LIN {X 0,Y 366.539,Z 659.329,A -85,B 0,C 180,E1 16261.22,E2 16261.22} C_VEL
LIN {X 0,Y 369.603,Z 643.731,A -85,B 0,C 180,E1 16259.522,E2 16259.522} C_VEL
LIN {X 0,Y 372.443,Z 626.719,A -85,B 0,C 180,E1 16258.031,E2 16258.031} C_VEL
LIN {X 0,Y 374.739,Z 609.542,A -85,B 0,C 180,E1 16256.842,E2 16256.842} C_VEL
LIN {X 0,Y 376.605,Z 590.744,A -85,B 0,C 180,E1 16255.852,E2 16255.852} C_VEL
LIN {X 0,Y 377.824,Z 571.243,A -85,B 0,C 180,E1 16255.127,E2 16255.127} C_VEL
LIN {X 0,Y 378.505,Z 547.045,A -85,B 0,C 180,E1 16254.58,E2 16254.58} C_VEL
LIN {X 0,Y 383.388,Z 388.518,A -85,B 0,C 180,E1 16251.66,E2 16251.66} C_VEL
LIN {X 0,Y 372.23,Z 368.985,A -85,B 0,C 180,E1 16249.629,E2 16249.629} C_VEL
LIN {X 0,Y 361.52,Z 352.259,A -85,B 0,C 180,E1 16247.541,E2 16247.541} C_VEL
LIN {X 0,Y 358.785,Z 347.938,A -85,B 0,C 180,E1 16246.899,E2 16246.899} C_VEL
LIN {X 0,Y 353.532,Z 335.825,A -85,B 0,C 180,E1 16243.861,E2 16243.861} C_VEL
LIN {X 0,Y 349.647,Z 327.602,A -85,B 0,C 180,E1 16241.563,E2 16241.563} C_VEL
LIN {X 0,Y 347.304,Z 322.978,A -85,B 0,C 180,E1 16240.157,E2 16240.157} C_VEL
LIN {X 0,Y 345.919,Z 319.541,A -85,B 0,C 180,E1 16239.059,E2 16239.059} C_VEL
LIN {X 0,Y 345.894,Z 319.384,A -85,B 0,C 180,E1 16234.823,E2 16234.823} C_VEL
LIN {X 0,Y 345.892,Z 319.382,A -85,B 0,C 180,E1 16230.527,E2 16230.527} C_VEL
LIN {X 0,Y 345.896,Z 319.388,A -85,B 0,C 180,E1 16226.354,E2 16226.354} C_VEL
LIN {X 0,Y 345.893,Z 319.4,A -85,B 0,C 180,E1 16222.252,E2 16222.252} C_VEL
LIN {X 0,Y 345.899,Z 319.385,A -85,B 0,C 180,E1 16218.014,E2 16218.014} C_VEL
LIN {X 0,Y 345.906,Z 319.366,A -85,B 0,C 180,E1 16213.785,E2 16213.785} C_VEL
LIN {X 0,Y 345.898,Z 319.37,A -85,B 0,C 180,E1 16209.484,E2 16209.484} C_VEL
LIN {X 0,Y 345.89,Z 319.398,A -85,B 0,C 180,E1 16205.308,E2 16205.308} C_VEL
LIN {X 0,Y 345.877,Z 319.386,A -85,B 0,C 180,E1 16201.16,E2 16201.16} C_VEL
LIN {X 0,Y 345.871,Z 319.369,A -85,B 0,C 180,E1 16197.018,E2 16197.018} C_VEL
LIN {X 0,Y 345.87,Z 319.378,A -85,B 0,C 180,E1 16192.86,E2 16192.86} C_VEL
LIN {X 0,Y 345.873,Z 319.401,A -85,B 0,C 180,E1 16188.664,E2 16188.664} C_VEL
LIN {X 0,Y 345.873,Z 319.4,A -85,B 0,C 180,E1 16184.405,E2 16184.405} C_VEL
LIN {X 0,Y 345.88,Z 319.39,A -85,B 0,C 180,E1 16180.056,E2 16180.056} C_VEL
LIN {X 0,Y 345.886,Z 319.384,A -85,B 0,C 180,E1 16175.947,E2 16175.947} C_VEL
LIN {X 0,Y 345.901,Z 319.385,A -85,B 0,C 180,E1 16171.702,E2 16171.702} C_VEL
LIN {X 0,Y 345.947,Z 319.628,A -85,B 0,C 180,E1 16169.507,E2 16169.507} C_VEL
LIN {X 0,Y 347.584,Z 323.392,A -85,B 0,C 180,E1 16168.43,E2 16168.43} C_VEL
LIN {X 0,Y 348.628,Z 324.913,A -85,B 0,C 180,E1 16167.956,E2 16167.956} C_VEL
LIN {X 0,Y 353.831,Z 334.918,A -85,B 0,C 180,E1 16165.39,E2 16165.39} C_VEL
LIN {X 0,Y 357.949,Z 342.981,A -85,B 0,C 180,E1 16163.49,E2 16163.49} C_VEL
LIN {X 0,Y 364.694,Z 357.152,A -85,B 0,C 180,E1 16160.502,E2 16160.502} C_VEL
LIN {X 0,Y 371.956,Z 374.258,A -85,B 0,C 180,E1 16157.359,E2 16157.359} C_VEL
LIN {X 0,Y 374.056,Z 379.335,A -85,B 0,C 180,E1 16156.557,E2 16156.557} C_VEL
LIN {X 0,Y 381.034,Z 392.431,A -85,B 0,C 180,E1 16155.246,E2 16155.246} C_VEL
LIN {X 0,Y 383.985,Z 429.126,A -85,B 0,C 180,E1 16153.918,E2 16153.918} C_VEL
LIN {X 0,Y 375.667,Z 632.493,A -85,B 0,C 180,E1 16149.71,E2 16149.71} C_VEL
LIN {X 0,Y 373.709,Z 654.478,A -85,B 0,C 180,E1 16149.004,E2 16149.004} C_VEL
LIN {X 0,Y 371.041,Z 675.386,A -85,B 0,C 180,E1 16148.054,E2 16148.054} C_VEL
LIN {X 0,Y 368.083,Z 694.62,A -85,B 0,C 180,E1 16146.892,E2 16146.892} C_VEL
LIN {X 0,Y 364.802,Z 713.742,A -85,B 0,C 180,E1 16145.427,E2 16145.427} C_VEL
LIN {X 0,Y 361.389,Z 732.08,A -85,B 0,C 180,E1 16143.691,E2 16143.691} C_VEL
LIN {X 0,Y 357.817,Z 750.227,A -85,B 0,C 180,E1 16141.596,E2 16141.596} C_VEL
LIN {X 0,Y 354.467,Z 767.276,A -85,B 0,C 180,E1 16139.207,E2 16139.207} C_VEL
LIN {X 0,Y 351.414,Z 783.149,A -85,B 0,C 180,E1 16136.531,E2 16136.531} C_VEL
LIN {X 0,Y 348.903,Z 797.366,A -85,B 0,C 180,E1 16133.653,E2 16133.653} C_VEL
LIN {X 0,Y 346.99,Z 809.978,A -85,B 0,C 180,E1 16130.581,E2 16130.581} C_VEL
LIN {X 0,Y 345.729,Z 820.44,A -85,B 0,C 180,E1 16127.503,E2 16127.503} C_VEL
LIN {X 0,Y 345.044,Z 829.017,A -85,B 0,C 180,E1 16124.43,E2 16124.43} C_VEL
LIN {X 0,Y 344.787,Z 836.104,A -85,B 0,C 180,E1 16121.203,E2 16121.203} C_VEL
LIN {X 0,Y 344.85,Z 841.123,A -85,B 0,C 180,E1 16118.167,E2 16118.167} C_VEL
LIN {X 0,Y 345.058,Z 844.743,A -85,B 0,C 180,E1 16114.987,E2 16114.987} C_VEL
LIN {X 0,Y 345.211,Z 846.508,A -85,B 0,C 180,E1 16112.158,E2 16112.158} C_VEL
LIN {X 0,Y 345.255,Z 846.827,A -85,B 0,C 180,E1 16109.17,E2 16109.17} C_VEL
LIN {X 0,Y 345.126,Z 845.656,A -85,B 0,C 180,E1 16106.179,E2 16106.179} C_VEL
LIN {X 0,Y 344.931,Z 842.863,A -85,B 0,C 180,E1 16103.175,E2 16103.175} C_VEL
LIN {X 0,Y 344.793,Z 838.223,A -85,B 0,C 180,E1 16099.98,E2 16099.98} C_VEL
LIN {X 0,Y 344.896,Z 831.799,A -85,B 0,C 180,E1 16096.761,E2 16096.761} C_VEL
LIN {X 0,Y 345.408,Z 823.997,A -85,B 0,C 180,E1 16093.693,E2 16093.693} C_VEL
LIN {X 0,Y 346.494,Z 813.722,A -85,B 0,C 180,E1 16090.444,E2 16090.444} C_VEL
LIN {X 0,Y 348.173,Z 801.841,A -85,B 0,C 180,E1 16087.369,E2 16087.369} C_VEL
LIN {X 0,Y 350.447,Z 788.441,A -85,B 0,C 180,E1 16084.481,E2 16084.481} C_VEL
LIN {X 0,Y 353.14,Z 774.009,A -85,B 0,C 180,E1 16081.874,E2 16081.874} C_VEL
LIN {X 0,Y 356.244,Z 758.161,A -85,B 0,C 180,E1 16079.47,E2 16079.47} C_VEL
LIN {X 0,Y 359.673,Z 740.767,A -85,B 0,C 180,E1 16077.27,E2 16077.27} C_VEL
LIN {X 0,Y 363.194,Z 722.371,A -85,B 0,C 180,E1 16075.356,E2 16075.356} C_VEL
LIN {X 0,Y 366.647,Z 702.966,A -85,B 0,C 180,E1 16073.719,E2 16073.719} C_VEL
LIN {X 0,Y 369.743,Z 683.735,A -85,B 0,C 180,E1 16072.426,E2 16072.426} C_VEL
LIN {X 0,Y 372.564,Z 663.659,A -85,B 0,C 180,E1 16071.389,E2 16071.389} C_VEL
LIN {X 0,Y 374.836,Z 642.783,A -85,B 0,C 180,E1 16070.598,E2 16070.598} C_VEL
LIN {X 0,Y 376.217,Z 620.758,A -85,B 0,C 180,E1 16070.027,E2 16070.027} C_VEL
LIN {X 0,Y 383.944,Z 427.198,A -85,B 0,C 180,E1 16066.047,E2 16066.047} C_VEL
LIN {X 0,Y 380.702,Z 391.532,A -85,B 0,C 180,E1 16064.711,E2 16064.711} C_VEL
LIN {X 0,Y 373.38,Z 377.914,A -85,B 0,C 180,E1 16063.277,E2 16063.277} C_VEL
LIN {X 0,Y 366.854,Z 362.006,A -85,B 0,C 180,E1 16060.441,E2 16060.441} C_VEL
LIN {X 0,Y 360.67,Z 348.666,A -85,B 0,C 180,E1 16057.782,E2 16057.782} C_VEL
LIN {X 0,Y 355.146,Z 337.373,A -85,B 0,C 180,E1 16055.25,E2 16055.25} C_VEL
LIN {X 0,Y 350.284,Z 328.233,A -85,B 0,C 180,E1 16052.947,E2 16052.947} C_VEL
LIN {X 0,Y 348.264,Z 324.159,A -85,B 0,C 180,E1 16051.888,E2 16051.888} C_VEL
LIN {X 0,Y 346.287,Z 320.952,A -85,B 0,C 180,E1 16050.927,E2 16050.927} C_VEL
LIN {X 0,Y 345.918,Z 319.456,A -85,B 0,C 180,E1 16050.413,E2 16050.413} C_VEL
LIN {X 0,Y 345.898,Z 319.385,A -85,B 0,C 180,E1 16046.248,E2 16046.248} C_VEL
LIN {X 0,Y 345.886,Z 319.383,A -85,B 0,C 180,E1 16042.073,E2 16042.073} C_VEL
LIN {X 0,Y 345.877,Z 319.378,A -85,B 0,C 180,E1 16037.844,E2 16037.844} C_VEL
LIN {X 0,Y 345.87,Z 319.372,A -85,B 0,C 180,E1 16033.542,E2 16033.542} C_VEL
LIN {X 0,Y 345.87,Z 319.379,A -85,B 0,C 180,E1 16029.316,E2 16029.316} C_VEL
LIN {X 0,Y 345.873,Z 319.402,A -85,B 0,C 180,E1 16025.141,E2 16025.141} C_VEL
LIN {X 0,Y 345.872,Z 319.39,A -85,B 0,C 180,E1 16020.993,E2 16020.993} C_VEL
LIN {X 0,Y 345.87,Z 319.369,A -85,B 0,C 180,E1 16016.851,E2 16016.851} C_VEL
LIN {X 0,Y 345.884,Z 319.379,A -85,B 0,C 180,E1 16012.692,E2 16012.692} C_VEL
LIN {X 0,Y 345.897,Z 319.401,A -85,B 0,C 180,E1 16008.491,E2 16008.491} C_VEL
LIN {X 0,Y 345.908,Z 319.379,A -85,B 0,C 180,E1 16004.234,E2 16004.234} C_VEL
LIN {X 0,Y 345.896,Z 319.37,A -85,B 0,C 180,E1 15999.956,E2 15999.956} C_VEL
LIN {X 0,Y 345.902,Z 319.373,A -85,B 0,C 180,E1 15995.947,E2 15995.947} C_VEL
LIN {X 0,Y 345.896,Z 319.385,A -85,B 0,C 180,E1 15991.701,E2 15991.701} C_VEL
LIN {X 0,Y 345.897,Z 319.393,A -85,B 0,C 180,E1 15987.569,E2 15987.569} C_VEL
LIN {X 0,Y 345.896,Z 319.393,A -85,B 0,C 180,E1 15983.453,E2 15983.453} C_VEL
LIN {X 0,Y 345.937,Z 319.68,A -85,B 0,C 180,E1 15980.73,E2 15980.73} C_VEL
LIN {X 0,Y 347.422,Z 323.162,A -85,B 0,C 180,E1 15979.643,E2 15979.643} C_VEL
LIN {X 0,Y 348.545,Z 325.55,A -85,B 0,C 180,E1 15978.934,E2 15978.934} C_VEL
LIN {X 0,Y 350.596,Z 329.771,A -85,B 0,C 180,E1 15977.697,E2 15977.697} C_VEL
LIN {X 0,Y 354.243,Z 337.521,A -85,B 0,C 180,E1 15975.568,E2 15975.568} C_VEL
LIN {X 0,Y 358.954,Z 348.373,A -85,B 0,C 180,E1 15972.896,E2 15972.896} C_VEL
LIN {X 0,Y 369.652,Z 364.898,A -85,B 0,C 180,E1 15970.738,E2 15970.738} C_VEL
LIN {X 0,Y 379.94,Z 382.361,A -85,B 0,C 180,E1 15968.834,E2 15968.834} C_VEL
LIN {X 0,Y 383.444,Z 389.074,A -85,B 0,C 180,E1 15968.206,E2 15968.206} C_VEL
LIN {X 0,Y 378.018,Z 564.942,A -85,B 0,C 180,E1 15964.946,E2 15964.946} C_VEL
LIN {X 0,Y 377.086,Z 583.644,A -85,B 0,C 180,E1 15964.345,E2 15964.345} C_VEL
LIN {X 0,Y 375.513,Z 601.927,A -85,B 0,C 180,E1 15963.496,E2 15963.496} C_VEL
LIN {X 0,Y 373.525,Z 618.693,A -85,B 0,C 180,E1 15962.458,E2 15962.458} C_VEL
LIN {X 0,Y 370.899,Z 636.019,A -85,B 0,C 180,E1 15961.094,E2 15961.094} C_VEL
LIN {X 0,Y 367.89,Z 652.482,A -85,B 0,C 180,E1 15959.466,E2 15959.466} C_VEL
LIN {X 0,Y 364.669,Z 667.723,A -85,B 0,C 180,E1 15957.604,E2 15957.604} C_VEL
LIN {X 0,Y 361.466,Z 681.388,A -85,B 0,C 180,E1 15955.563,E2 15955.563} C_VEL
LIN {X 0,Y 358.145,Z 694.464,A -85,B 0,C 180,E1 15953.18,E2 15953.18} C_VEL
LIN {X 0,Y 355.074,Z 705.939,A -85,B 0,C 180,E1 15950.608,E2 15950.608} C_VEL
LIN {X 0,Y 352.38,Z 715.885,A -85,B 0,C 180,E1 15947.845,E2 15947.845} C_VEL
LIN {X 0,Y 350.093,Z 724.318,A -85,B 0,C 180,E1 15944.894,E2 15944.894} C_VEL
LIN {X 0,Y 348.354,Z 731.066,A -85,B 0,C 180,E1 15941.831,E2 15941.831} C_VEL
LIN {X 0,Y 347.117,Z 736.256,A -85,B 0,C 180,E1 15938.614,E2 15938.614} C_VEL
LIN {X 0,Y 346.367,Z 739.644,A -85,B 0,C 180,E1 15935.466,E2 15935.466} C_VEL
LIN {X 0,Y 345.992,Z 741.548,A -85,B 0,C 180,E1 15932.153,E2 15932.153} C_VEL
LIN {X 0,Y 345.939,Z 741.818,A -85,B 0,C 180,E1 15928.841,E2 15928.841} C_VEL
LIN {X 0,Y 346.204,Z 740.465,A -85,B 0,C 180,E1 15925.528,E2 15925.528} C_VEL
LIN {X 0,Y 346.714,Z 738.05,A -85,B 0,C 180,E1 15922.764,E2 15922.764} C_VEL
LIN {X 0,Y 346.061,Z 736.752,A -85,B 0,C 180,E1 15921.504,E2 15921.504} C_VEL
LIN {X 0,Y 341.253,Z 732.89,A -85,B 0,C 180,E1 15918.207,E2 15918.207} C_VEL
LIN {X 0,Y 340.994,Z 730.849,A -85,B 0,C 180,E1 15917.039,E2 15917.039} C_VEL
LIN {X 0,Y 342.986,Z 723.691,A -85,B 0,C 180,E1 15913.923,E2 15913.923} C_VEL
LIN {X 0,Y 345.546,Z 714.785,A -85,B 0,C 180,E1 15910.916,E2 15910.916} C_VEL
LIN {X 0,Y 348.539,Z 704.306,A -85,B 0,C 180,E1 15908.104,E2 15908.104} C_VEL
LIN {X 0,Y 351.909,Z 692.224,A -85,B 0,C 180,E1 15905.493,E2 15905.493} C_VEL
LIN {X 0,Y 355.499,Z 678.411,A -85,B 0,C 180,E1 15903.076,E2 15903.076} C_VEL
LIN {X 0,Y 358.999,Z 663.723,A -85,B 0,C 180,E1 15900.99,E2 15900.99} C_VEL
LIN {X 0,Y 362.256,Z 648.294,A -85,B 0,C 180,E1 15899.204,E2 15899.204} C_VEL
LIN {X 0,Y 365.281,Z 631.623,A -85,B 0,C 180,E1 15897.648,E2 15897.648} C_VEL
LIN {X 0,Y 367.892,Z 613.759,A -85,B 0,C 180,E1 15896.33,E2 15896.33} C_VEL
LIN {X 0,Y 369.927,Z 595.416,A -85,B 0,C 180,E1 15895.295,E2 15895.295} C_VEL
LIN {X 0,Y 371.317,Z 576.435,A -85,B 0,C 180,E1 15894.519,E2 15894.519} C_VEL
LIN {X 0,Y 372.031,Z 556.598,A -85,B 0,C 180,E1 15893.998,E2 15893.998} C_VEL
LIN {X 0,Y 377.33,Z 391.658,A -85,B 0,C 180,E1 15890.912,E2 15890.912} C_VEL
LIN {X 0,Y 366.892,Z 373.263,A -85,B 0,C 180,E1 15888.936,E2 15888.936} C_VEL
LIN {X 0,Y 356.62,Z 357.168,A -85,B 0,C 180,E1 15886.859,E2 15886.859} C_VEL
LIN {X 0,Y 351.137,Z 348.844,A -85,B 0,C 180,E1 15885.621,E2 15885.621} C_VEL
LIN {X 0,Y 345.873,Z 337.173,A -85,B 0,C 180,E1 15882.512,E2 15882.512} C_VEL
LIN {X 0,Y 341.765,Z 328.63,A -85,B 0,C 180,E1 15879.961,E2 15879.961} C_VEL
LIN {X 0,Y 339.688,Z 324.424,A -85,B 0,C 180,E1 15878.61,E2 15878.61} C_VEL
LIN {X 0,Y 337.986,Z 320.54,A -85,B 0,C 180,E1 15877.273,E2 15877.273} C_VEL
LIN {X 0,Y 337.951,Z 320.371,A -85,B 0,C 180,E1 15872.983,E2 15872.983} C_VEL
LIN {X 0,Y 337.95,Z 320.368,A -85,B 0,C 180,E1 15868.64,E2 15868.64} C_VEL
LIN {X 0,Y 337.952,Z 320.361,A -85,B 0,C 180,E1 15864.326,E2 15864.326} C_VEL
LIN {X 0,Y 337.949,Z 320.361,A -85,B 0,C 180,E1 15860.253,E2 15860.253} C_VEL
LIN {X 0,Y 337.96,Z 320.373,A -85,B 0,C 180,E1 15855.953,E2 15855.953} C_VEL
LIN {X 0,Y 337.964,Z 320.385,A -85,B 0,C 180,E1 15851.699,E2 15851.699} C_VEL
LIN {X 0,Y 337.964,Z 320.361,A -85,B 0,C 180,E1 15847.48,E2 15847.48} C_VEL
LIN {X 0,Y 337.939,Z 320.356,A -85,B 0,C 180,E1 15843.223,E2 15843.223} C_VEL
LIN {X 0,Y 337.929,Z 320.376,A -85,B 0,C 180,E1 15838.983,E2 15838.983} C_VEL
LIN {X 0,Y 337.927,Z 320.39,A -85,B 0,C 180,E1 15834.738,E2 15834.738} C_VEL
LIN {X 0,Y 337.926,Z 320.37,A -85,B 0,C 180,E1 15830.463,E2 15830.463} C_VEL
LIN {X 0,Y 337.932,Z 320.361,A -85,B 0,C 180,E1 15826.134,E2 15826.134} C_VEL
LIN {X 0,Y 337.943,Z 320.364,A -85,B 0,C 180,E1 15821.901,E2 15821.901} C_VEL
LIN {X 0,Y 337.955,Z 320.368,A -85,B 0,C 180,E1 15817.748,E2 15817.748} C_VEL
LIN {X 0,Y 337.969,Z 320.367,A -85,B 0,C 180,E1 15813.467,E2 15813.467} C_VEL
LIN {X 0,Y 338.026,Z 320.649,A -85,B 0,C 180,E1 15811.307,E2 15811.307} C_VEL
LIN {X 0,Y 339.317,Z 323.956,A -85,B 0,C 180,E1 15810.328,E2 15810.328} C_VEL
LIN {X 0,Y 340.859,Z 326.12,A -85,B 0,C 180,E1 15809.585,E2 15809.585} C_VEL
LIN {X 0,Y 342.798,Z 329.791,A -85,B 0,C 180,E1 15808.527,E2 15808.527} C_VEL
LIN {X 0,Y 348.279,Z 340.218,A -85,B 0,C 180,E1 15805.758,E2 15805.758} C_VEL
LIN {X 0,Y 354.382,Z 352.579,A -85,B 0,C 180,E1 15802.859,E2 15802.859} C_VEL
LIN {X 0,Y 360.708,Z 366.49,A -85,B 0,C 180,E1 15799.978,E2 15799.978} C_VEL
LIN {X 0,Y 365.81,Z 378.592,A -85,B 0,C 180,E1 15797.802,E2 15797.802} C_VEL
LIN {X 0,Y 375.242,Z 395.721,A -85,B 0,C 180,E1 15795.957,E2 15795.957} C_VEL
LIN {X 0,Y 377.885,Z 430.233,A -85,B 0,C 180,E1 15794.686,E2 15794.686} C_VEL
LIN {X 0,Y 369.297,Z 631.618,A -85,B 0,C 180,E1 15790.468,E2 15790.468} C_VEL
LIN {X 0,Y 367.272,Z 653.63,A -85,B 0,C 180,E1 15789.753,E2 15789.753} C_VEL
LIN {X 0,Y 364.435,Z 674.971,A -85,B 0,C 180,E1 15788.771,E2 15788.771} C_VEL
LIN {X 0,Y 361.176,Z 695.239,A -85,B 0,C 180,E1 15787.518,E2 15787.518} C_VEL
LIN {X 0,Y 357.602,Z 714.966,A -85,B 0,C 180,E1 15785.955,E2 15785.955} C_VEL
LIN {X 0,Y 353.991,Z 733.289,A -85,B 0,C 180,E1 15784.149,E2 15784.149} C_VEL
LIN {X 0,Y 350.491,Z 750.079,A -85,B 0,C 180,E1 15782.142,E2 15782.142} C_VEL
LIN {X 0,Y 347.071,Z 766.57,A -85,B 0,C 180,E1 15779.772,E2 15779.772} C_VEL
LIN {X 0,Y 343.961,Z 781.792,A -85,B 0,C 180,E1 15777.153,E2 15777.153} C_VEL
LIN {X 0,Y 341.276,Z 796.036,A -85,B 0,C 180,E1 15774.215,E2 15774.215} C_VEL
LIN {X 0,Y 339.307,Z 808.039,A -85,B 0,C 180,E1 15771.25,E2 15771.25} C_VEL
LIN {X 0,Y 337.908,Z 818.643,A -85,B 0,C 180,E1 15768.1,E2 15768.1} C_VEL
LIN {X 0,Y 337.111,Z 827.752,A -85,B 0,C 180,E1 15764.777,E2 15764.777} C_VEL
LIN {X 0,Y 336.824,Z 834.857,A -85,B 0,C 180,E1 15761.472,E2 15761.472} C_VEL
LIN {X 0,Y 336.893,Z 839.896,A -85,B 0,C 180,E1 15758.362,E2 15758.362} C_VEL
LIN {X 0,Y 337.125,Z 843.531,A -85,B 0,C 180,E1 15755.104,E2 15755.104} C_VEL
LIN {X 0,Y 337.296,Z 845.304,A -85,B 0,C 180,E1 15752.208,E2 15752.208} C_VEL
LIN {X 0,Y 337.344,Z 845.625,A -85,B 0,C 180,E1 15749.151,E2 15749.151} C_VEL
LIN {X 0,Y 337.2,Z 844.447,A -85,B 0,C 180,E1 15746.09,E2 15746.09} C_VEL
LIN {X 0,Y 336.979,Z 841.641,A -85,B 0,C 180,E1 15743.013,E2 15743.013} C_VEL
LIN {X 0,Y 336.832,Z 836.984,A -85,B 0,C 180,E1 15739.741,E2 15739.741} C_VEL
LIN {X 0,Y 336.947,Z 830.538,A -85,B 0,C 180,E1 15736.443,E2 15736.443} C_VEL
LIN {X 0,Y 337.497,Z 822.711,A -85,B 0,C 180,E1 15733.3,E2 15733.3} C_VEL
LIN {X 0,Y 338.683,Z 812.419,A -85,B 0,C 180,E1 15729.974,E2 15729.974} C_VEL
LIN {X 0,Y 340.528,Z 800.34,A -85,B 0,C 180,E1 15726.784,E2 15726.784} C_VEL
LIN {X 0,Y 342.929,Z 787.093,A -85,B 0,C 180,E1 15723.88,E2 15723.88} C_VEL
LIN {X 0,Y 345.7,Z 773.129,A -85,B 0,C 180,E1 15721.308,E2 15721.308} C_VEL
LIN {X 0,Y 348.97,Z 757.336,A -85,B 0,C 180,E1 15718.859,E2 15718.859} C_VEL
LIN {X 0,Y 352.569,Z 740.004,A -85,B 0,C 180,E1 15716.622,E2 15716.622} C_VEL
LIN {X 0,Y 356.261,Z 721.682,A -85,B 0,C 180,E1 15714.681,E2 15714.681} C_VEL
LIN {X 0,Y 359.684,Z 703.397,A -85,B 0,C 180,E1 15713.1,E2 15713.1} C_VEL
LIN {X 0,Y 362.893,Z 684.551,A -85,B 0,C 180,E1 15711.791,E2 15711.791} C_VEL
LIN {X 0,Y 365.952,Z 663.876,A -85,B 0,C 180,E1 15710.69,E2 15710.69} C_VEL
LIN {X 0,Y 368.407,Z 642.256,A -85,B 0,C 180,E1 15709.855,E2 15709.855} C_VEL
LIN {X 0,Y 369.854,Z 620.163,A -85,B 0,C 180,E1 15709.272,E2 15709.272} C_VEL
LIN {X 0,Y 377.84,Z 428.2,A -85,B 0,C 180,E1 15705.277,E2 15705.277} C_VEL
LIN {X 0,Y 374.987,Z 395.198,A -85,B 0,C 180,E1 15704.021,E2 15704.021} C_VEL
LIN {X 0,Y 365.339,Z 377.727,A -85,B 0,C 180,E1 15702.106,E2 15702.106} C_VEL
LIN {X 0,Y 358.592,Z 361.64,A -85,B 0,C 180,E1 15699.061,E2 15699.061} C_VEL
LIN {X 0,Y 351.937,Z 347.377,A -85,B 0,C 180,E1 15696.021,E2 15696.021} C_VEL
LIN {X 0,Y 346.773,Z 337.483,A -85,B 0,C 180,E1 15693.565,E2 15693.565} C_VEL
LIN {X 0,Y 344.569,Z 333.342,A -85,B 0,C 180,E1 15692.468,E2 15692.468} C_VEL
LIN {X 0,Y 342.71,Z 329.695,A -85,B 0,C 180,E1 15691.482,E2 15691.482} C_VEL
LIN {X 0,Y 340.761,Z 325.802,A -85,B 0,C 180,E1 15690.387,E2 15690.387} C_VEL
LIN {X 0,Y 338.388,Z 322.126,A -85,B 0,C 180,E1 15689.178,E2 15689.178} C_VEL
LIN {X 0,Y 338,Z 320.488,A -85,B 0,C 180,E1 15688.634,E2 15688.634} C_VEL
LIN {X 0,Y 337.962,Z 320.376,A -85,B 0,C 180,E1 15684.33,E2 15684.33} C_VEL
LIN {X 0,Y 337.957,Z 320.383,A -85,B 0,C 180,E1 15680.252,E2 15680.252} C_VEL
LIN {X 0,Y 337.942,Z 320.391,A -85,B 0,C 180,E1 15675.942,E2 15675.942} C_VEL
LIN {X 0,Y 337.932,Z 320.383,A -85,B 0,C 180,E1 15671.607,E2 15671.607} C_VEL
LIN {X 0,Y 337.928,Z 320.366,A -85,B 0,C 180,E1 15667.309,E2 15667.309} C_VEL
LIN {X 0,Y 337.93,Z 320.359,A -85,B 0,C 180,E1 15663.053,E2 15663.053} C_VEL
LIN {X 0,Y 337.931,Z 320.38,A -85,B 0,C 180,E1 15658.982,E2 15658.982} C_VEL
LIN {X 0,Y 337.943,Z 320.386,A -85,B 0,C 180,E1 15654.737,E2 15654.737} C_VEL
LIN {X 0,Y 337.954,Z 320.359,A -85,B 0,C 180,E1 15650.463,E2 15650.463} C_VEL
LIN {X 0,Y 337.957,Z 320.356,A -85,B 0,C 180,E1 15646.134,E2 15646.134} C_VEL
LIN {X 0,Y 337.951,Z 320.374,A -85,B 0,C 180,E1 15641.901,E2 15641.901} C_VEL
LIN {X 0,Y 337.951,Z 320.389,A -85,B 0,C 180,E1 15637.746,E2 15637.746} C_VEL
LIN {X 0,Y 337.946,Z 320.38,A -85,B 0,C 180,E1 15633.464,E2 15633.464} C_VEL
LIN {X 0,Y 337.945,Z 320.375,A -85,B 0,C 180,E1 15629.213,E2 15629.213} C_VEL
LIN {X 0,Y 337.949,Z 320.375,A -85,B 0,C 180,E1 15624.972,E2 15624.972} C_VEL
LIN {X 0,Y 338.009,Z 320.663,A -85,B 0,C 180,E1 15622.511,E2 15622.511} C_VEL
LIN {X 0,Y 339.793,Z 324.568,A -85,B 0,C 180,E1 15621.188,E2 15621.188} C_VEL
LIN {X 0,Y 342.825,Z 330.891,A -85,B 0,C 180,E1 15619.208,E2 15619.208} C_VEL
LIN {X 0,Y 346.651,Z 338.868,A -85,B 0,C 180,E1 15616.875,E2 15616.875} C_VEL
LIN {X 0,Y 351.508,Z 349.594,A -85,B 0,C 180,E1 15614.12,E2 15614.12} C_VEL
LIN {X 0,Y 362.352,Z 366.047,A -85,B 0,C 180,E1 15611.838,E2 15611.838} C_VEL
LIN {X 0,Y 373.097,Z 384.003,A -85,B 0,C 180,E1 15609.754,E2 15609.754} C_VEL
LIN {X 0,Y 377.371,Z 392.19,A -85,B 0,C 180,E1 15608.955,E2 15608.955} C_VEL
LIN {X 0,Y 371.728,Z 565.463,A -85,B 0,C 180,E1 15605.698,E2 15605.698} C_VEL
LIN {X 0,Y 370.761,Z 584.169,A -85,B 0,C 180,E1 15605.093,E2 15605.093} C_VEL
LIN {X 0,Y 369.14,Z 602.364,A -85,B 0,C 180,E1 15604.243,E2 15604.243} C_VEL
LIN {X 0,Y 366.924,Z 620.305,A -85,B 0,C 180,E1 15603.116,E2 15603.116} C_VEL
LIN {X 0,Y 364.314,Z 636.765,A -85,B 0,C 180,E1 15601.798,E2 15601.798} C_VEL
LIN {X 0,Y 361.195,Z 653.169,A -85,B 0,C 180,E1 15600.16,E2 15600.16} C_VEL
LIN {X 0,Y 357.832,Z 668.479,A -85,B 0,C 180,E1 15598.269,E2 15598.269} C_VEL
LIN {X 0,Y 354.354,Z 682.686,A -85,B 0,C 180,E1 15596.114,E2 15596.114} C_VEL
LIN {X 0,Y 351.104,Z 694.934,A -85,B 0,C 180,E1 15593.852,E2 15593.852} C_VEL
LIN {X 0,Y 347.854,Z 706.532,A -85,B 0,C 180,E1 15591.233,E2 15591.233} C_VEL
LIN {X 0,Y 344.99,Z 716.587,A -85,B 0,C 180,E1 15588.415,E2 15588.415} C_VEL
LIN {X 0,Y 342.551,Z 725.119,A -85,B 0,C 180,E1 15585.403,E2 15585.403} C_VEL
LIN {X 0,Y 340.64,Z 732.111,A -85,B 0,C 180,E1 15582.194,E2 15582.194} C_VEL
LIN {X 0,Y 339.338,Z 737.236,A -85,B 0,C 180,E1 15578.984,E2 15578.984} C_VEL
LIN {X 0,Y 338.486,Z 740.849,A -85,B 0,C 180,E1 15575.594,E2 15575.594} C_VEL
LIN {X 0,Y 338.087,Z 742.75,A -85,B 0,C 180,E1 15572.203,E2 15572.203} C_VEL
LIN {X 0,Y 338.031,Z 743.019,A -85,B 0,C 180,E1 15568.814,E2 15568.814} C_VEL
LIN {X 0,Y 338.314,Z 741.668,A -85,B 0,C 180,E1 15565.423,E2 15565.423} C_VEL
LIN {X 0,Y 339.006,Z 738.638,A -85,B 0,C 180,E1 15562.032,E2 15562.032} C_VEL
LIN {X 0,Y 340.139,Z 734.091,A -85,B 0,C 180,E1 15558.813,E2 15558.813} C_VEL
LIN {X 0,Y 340.994,Z 730.849,A -85,B 0,C 180,E1 15557.039,E2 15557.039} C_VEL
LIN {X 0,Y 340.753,Z 728.553,A -85,B 0,C 180,E1 15555.793,E2 15555.793} C_VEL
LIN {X 0,Y 337.133,Z 722.237,A -85,B 0,C 180,E1 15552.617,E2 15552.617} C_VEL
LIN {X 0,Y 337.17,Z 718.967,A -85,B 0,C 180,E1 15551.419,E2 15551.419} C_VEL
LIN {X 0,Y 340.019,Z 709.487,A -85,B 0,C 180,E1 15548.616,E2 15548.616} C_VEL
LIN {X 0,Y 343.339,Z 698.274,A -85,B 0,C 180,E1 15545.94,E2 15545.94} C_VEL
LIN {X 0,Y 346.919,Z 685.521,A -85,B 0,C 180,E1 15543.467,E2 15543.467} C_VEL
LIN {X 0,Y 350.51,Z 671.669,A -85,B 0,C 180,E1 15541.272,E2 15541.272} C_VEL
LIN {X 0,Y 353.941,Z 657.099,A -85,B 0,C 180,E1 15539.382,E2 15539.382} C_VEL
LIN {X 0,Y 357.224,Z 641.016,A -85,B 0,C 180,E1 15537.684,E2 15537.684} C_VEL
LIN {X 0,Y 360.105,Z 624.301,A -85,B 0,C 180,E1 15536.269,E2 15536.269} C_VEL
LIN {X 0,Y 362.509,Z 606.576,A -85,B 0,C 180,E1 15535.089,E2 15535.089} C_VEL
LIN {X 0,Y 364.381,Z 587.477,A -85,B 0,C 180,E1 15534.139,E2 15534.139} C_VEL
LIN {X 0,Y 365.522,Z 567.969,A -85,B 0,C 180,E1 15533.47,E2 15533.47} C_VEL
LIN {X 0,Y 367.419,Z 507.657,A -85,B 0,C 180,E1 15532.283,E2 15532.283} C_VEL
LIN {X 0,Y 371.29,Z 394.593,A -85,B 0,C 180,E1 15530.129,E2 15530.129} C_VEL
LIN {X 0,Y 360.772,Z 376.206,A -85,B 0,C 180,E1 15528.055,E2 15528.055} C_VEL
LIN {X 0,Y 350.107,Z 359.514,A -85,B 0,C 180,E1 15525.793,E2 15525.793} C_VEL
LIN {X 0,Y 343.368,Z 349.702,A -85,B 0,C 180,E1 15524.22,E2 15524.22} C_VEL
LIN {X 0,Y 338.518,Z 338.884,A -85,B 0,C 180,E1 15521.198,E2 15521.198} C_VEL
LIN {X 0,Y 334.18,Z 330.098,A -85,B 0,C 180,E1 15518.383,E2 15518.383} C_VEL
LIN {X 0,Y 331.916,Z 325.62,A -85,B 0,C 180,E1 15516.832,E2 15516.832} C_VEL
LIN {X 0,Y 330.164,Z 322.103,A -85,B 0,C 180,E1 15515.553,E2 15515.553} C_VEL
LIN {X 0,Y 330.019,Z 321.371,A -85,B 0,C 180,E1 15514.933,E2 15514.933} C_VEL
LIN {X 0,Y 330.012,Z 321.359,A -85,B 0,C 180,E1 15510.598,E2 15510.598} C_VEL
LIN {X 0,Y 330.014,Z 321.367,A -85,B 0,C 180,E1 15506.448,E2 15506.448} C_VEL
LIN {X 0,Y 330.027,Z 321.377,A -85,B 0,C 180,E1 15502.066,E2 15502.066} C_VEL
LIN {X 0,Y 330.032,Z 321.367,A -85,B 0,C 180,E1 15497.636,E2 15497.636} C_VEL
LIN {X 0,Y 330.013,Z 321.348,A -85,B 0,C 180,E1 15493.313,E2 15493.313} C_VEL
LIN {X 0,Y 329.992,Z 321.345,A -85,B 0,C 180,E1 15488.984,E2 15488.984} C_VEL
LIN {X 0,Y 329.984,Z 321.366,A -85,B 0,C 180,E1 15484.693,E2 15484.693} C_VEL
LIN {X 0,Y 329.979,Z 321.379,A -85,B 0,C 180,E1 15480.348,E2 15480.348} C_VEL
LIN {X 0,Y 329.988,Z 321.354,A -85,B 0,C 180,E1 15476.004,E2 15476.004} C_VEL
LIN {X 0,Y 330.001,Z 321.346,A -85,B 0,C 180,E1 15471.813,E2 15471.813} C_VEL
LIN {X 0,Y 330.018,Z 321.353,A -85,B 0,C 180,E1 15467.578,E2 15467.578} C_VEL
LIN {X 0,Y 330.031,Z 321.366,A -85,B 0,C 180,E1 15463.273,E2 15463.273} C_VEL
LIN {X 0,Y 330.021,Z 321.374,A -85,B 0,C 180,E1 15458.867,E2 15458.867} C_VEL
LIN {X 0,Y 330.018,Z 321.377,A -85,B 0,C 180,E1 15454.711,E2 15454.711} C_VEL
LIN {X 0,Y 330.082,Z 321.657,A -85,B 0,C 180,E1 15453.325,E2 15453.325} C_VEL
LIN {X 0,Y 331.592,Z 325.229,A -85,B 0,C 180,E1 15452.136,E2 15452.136} C_VEL
LIN {X 0,Y 332.907,Z 326.905,A -85,B 0,C 180,E1 15451.475,E2 15451.475} C_VEL
LIN {X 0,Y 334.885,Z 330.792,A -85,B 0,C 180,E1 15450.29,E2 15450.29} C_VEL
LIN {X 0,Y 336.066,Z 333.043,A -85,B 0,C 180,E1 15449.617,E2 15449.617} C_VEL
LIN {X 0,Y 338.831,Z 338.21,A -85,B 0,C 180,E1 15448.116,E2 15448.116} C_VEL
LIN {X 0,Y 344.725,Z 349.404,A -85,B 0,C 180,E1 15445.153,E2 15445.153} C_VEL
LIN {X 0,Y 351.794,Z 364.539,A -85,B 0,C 180,E1 15441.714,E2 15441.714} C_VEL
LIN {X 0,Y 357.569,Z 377.862,A -85,B 0,C 180,E1 15439.132,E2 15439.132} C_VEL
LIN {X 0,Y 368.259,Z 396.802,A -85,B 0,C 180,E1 15436.934,E2 15436.934} C_VEL
LIN {X 0,Y 369.574,Z 399.796,A -85,B 0,C 180,E1 15436.66,E2 15436.66} C_VEL
LIN {X 0,Y 371.855,Z 431.34,A -85,B 0,C 180,E1 15435.478,E2 15435.478} C_VEL
LIN {X 0,Y 362.986,Z 630.851,A -85,B 0,C 180,E1 15431.25,E2 15431.25} C_VEL
LIN {X 0,Y 360.899,Z 652.81,A -85,B 0,C 180,E1 15430.527,E2 15430.527} C_VEL
LIN {X 0,Y 357.99,Z 673.843,A -85,B 0,C 180,E1 15429.552,E2 15429.552} C_VEL
LIN {X 0,Y 354.589,Z 694.236,A -85,B 0,C 180,E1 15428.28,E2 15428.28} C_VEL
LIN {X 0,Y 350.954,Z 713.405,A -85,B 0,C 180,E1 15426.746,E2 15426.746} C_VEL
LIN {X 0,Y 347.238,Z 731.415,A -85,B 0,C 180,E1 15424.959,E2 15424.959} C_VEL
LIN {X 0,Y 343.48,Z 748.656,A -85,B 0,C 180,E1 15422.88,E2 15422.88} C_VEL
LIN {X 0,Y 339.836,Z 765.3,A -85,B 0,C 180,E1 15420.452,E2 15420.452} C_VEL
LIN {X 0,Y 336.55,Z 780.44,A -85,B 0,C 180,E1 15417.802,E2 15417.802} C_VEL
LIN {X 0,Y 333.831,Z 793.946,A -85,B 0,C 180,E1 15414.98,E2 15414.98} C_VEL
LIN {X 0,Y 331.667,Z 806.101,A -85,B 0,C 180,E1 15411.95,E2 15411.95} C_VEL
LIN {X 0,Y 330.113,Z 816.843,A -85,B 0,C 180,E1 15408.726,E2 15408.726} C_VEL
LIN {X 0,Y 329.206,Z 826.04,A -85,B 0,C 180,E1 15405.321,E2 15405.321} C_VEL
LIN {X 0,Y 328.863,Z 833.265,A -85,B 0,C 180,E1 15401.931,E2 15401.931} C_VEL
LIN {X 0,Y 328.935,Z 838.668,A -85,B 0,C 180,E1 15398.565,E2 15398.565} C_VEL
LIN {X 0,Y 329.19,Z 842.319,A -85,B 0,C 180,E1 15395.228,E2 15395.228} C_VEL
LIN {X 0,Y 329.381,Z 844.1,A -85,B 0,C 180,E1 15392.262,E2 15392.262} C_VEL
LIN {X 0,Y 329.434,Z 844.424,A -85,B 0,C 180,E1 15389.13,E2 15389.13} C_VEL
LIN {X 0,Y 329.272,Z 843.237,A -85,B 0,C 180,E1 15385.995,E2 15385.995} C_VEL
LIN {X 0,Y 329.027,Z 840.42,A -85,B 0,C 180,E1 15382.843,E2 15382.843} C_VEL
LIN {X 0,Y 328.865,Z 835.744,A -85,B 0,C 180,E1 15379.49,E2 15379.49} C_VEL
LIN {X 0,Y 329.002,Z 829.277,A -85,B 0,C 180,E1 15376.109,E2 15376.109} C_VEL
LIN {X 0,Y 329.612,Z 821.315,A -85,B 0,C 180,E1 15372.848,E2 15372.848} C_VEL
LIN {X 0,Y 330.897,Z 811.117,A -85,B 0,C 180,E1 15369.482,E2 15369.482} C_VEL
LIN {X 0,Y 332.85,Z 799.201,A -85,B 0,C 180,E1 15366.264,E2 15366.264} C_VEL
LIN {X 0,Y 335.449,Z 785.75,A -85,B 0,C 180,E1 15363.252,E2 15363.252} C_VEL
LIN {X 0,Y 338.62,Z 770.765,A -85,B 0,C 180,E1 15360.456,E2 15360.456} C_VEL
LIN {X 0,Y 341.998,Z 755.34,A -85,B 0,C 180,E1 15358.052,E2 15358.052} C_VEL
LIN {X 0,Y 345.669,Z 738.547,A -85,B 0,C 180,E1 15355.866,E2 15355.866} C_VEL
LIN {X 0,Y 349.551,Z 720.157,A -85,B 0,C 180,E1 15353.898,E2 15353.898} C_VEL
LIN {X 0,Y 353.319,Z 700.736,A -85,B 0,C 180,E1 15352.218,E2 15352.218} C_VEL
LIN {X 0,Y 356.709,Z 681.467,A -85,B 0,C 180,E1 15350.901,E2 15350.901} C_VEL
LIN {X 0,Y 359.711,Z 661.609,A -85,B 0,C 180,E1 15349.858,E2 15349.858} C_VEL
LIN {X 0,Y 362.13,Z 640.669,A -85,B 0,C 180,E1 15349.053,E2 15349.053} C_VEL
LIN {X 0,Y 363.596,Z 618.696,A -85,B 0,C 180,E1 15348.472,E2 15348.472} C_VEL
LIN {X 0,Y 371.808,Z 429.248,A -85,B 0,C 180,E1 15344.483,E2 15344.483} C_VEL
LIN {X 0,Y 369.242,Z 398.809,A -85,B 0,C 180,E1 15343.296,E2 15343.296} C_VEL
LIN {X 0,Y 359.659,Z 381.559,A -85,B 0,C 180,E1 15341.345,E2 15341.345} C_VEL
LIN {X 0,Y 357.005,Z 376.819,A -85,B 0,C 180,E1 15340.734,E2 15340.734} C_VEL
LIN {X 0,Y 350.035,Z 360.556,A -85,B 0,C 180,E1 15337.432,E2 15337.432} C_VEL
LIN {X 0,Y 343.951,Z 348.039,A -85,B 0,C 180,E1 15334.531,E2 15334.531} C_VEL
LIN {X 0,Y 339.399,Z 339.27,A -85,B 0,C 180,E1 15332.223,E2 15332.223} C_VEL
LIN {X 0,Y 337.08,Z 334.954,A -85,B 0,C 180,E1 15330.994,E2 15330.994} C_VEL
LIN {X 0,Y 335.156,Z 331.101,A -85,B 0,C 180,E1 15329.881,E2 15329.881} C_VEL
LIN {X 0,Y 333.053,Z 327.414,A -85,B 0,C 180,E1 15328.707,E2 15328.707} C_VEL
LIN {X 0,Y 332.535,Z 326.256,A -85,B 0,C 180,E1 15328.364,E2 15328.364} C_VEL
LIN {X 0,Y 330.422,Z 323.03,A -85,B 0,C 180,E1 15327.189,E2 15327.189} C_VEL
LIN {X 0,Y 330.046,Z 321.433,A -85,B 0,C 180,E1 15326.581,E2 15326.581} C_VEL
LIN {X 0,Y 330.017,Z 321.356,A -85,B 0,C 180,E1 15322.254,E2 15322.254} C_VEL
LIN {X 0,Y 330.003,Z 321.353,A -85,B 0,C 180,E1 15317.947,E2 15317.947} C_VEL
LIN {X 0,Y 329.993,Z 321.349,A -85,B 0,C 180,E1 15313.67,E2 15313.67} C_VEL
LIN {X 0,Y 329.991,Z 321.356,A -85,B 0,C 180,E1 15309.417,E2 15309.417} C_VEL
LIN {X 0,Y 329.993,Z 321.38,A -85,B 0,C 180,E1 15305.215,E2 15305.215} C_VEL
LIN {X 0,Y 330.002,Z 321.367,A -85,B 0,C 180,E1 15300.868,E2 15300.868} C_VEL
LIN {X 0,Y 330.005,Z 321.345,A -85,B 0,C 180,E1 15296.504,E2 15296.504} C_VEL
LIN {X 0,Y 330.01,Z 321.346,A -85,B 0,C 180,E1 15292.163,E2 15292.163} C_VEL
LIN {X 0,Y 330.002,Z 321.376,A -85,B 0,C 180,E1 15287.932,E2 15287.932} C_VEL
LIN {X 0,Y 329.999,Z 321.371,A -85,B 0,C 180,E1 15283.633,E2 15283.633} C_VEL
LIN {X 0,Y 329.996,Z 321.355,A -85,B 0,C 180,E1 15279.237,E2 15279.237} C_VEL
LIN {X 0,Y 330.003,Z 321.349,A -85,B 0,C 180,E1 15274.901,E2 15274.901} C_VEL
LIN {X 0,Y 330.014,Z 321.352,A -85,B 0,C 180,E1 15270.755,E2 15270.755} C_VEL
LIN {X 0,Y 330.024,Z 321.355,A -85,B 0,C 180,E1 15266.537,E2 15266.537} C_VEL
LIN {X 0,Y 330.063,Z 321.623,A -85,B 0,C 180,E1 15264.507,E2 15264.507} C_VEL
LIN {X 0,Y 331.69,Z 325.358,A -85,B 0,C 180,E1 15263.139,E2 15263.139} C_VEL
LIN {X 0,Y 332.674,Z 327.051,A -85,B 0,C 180,E1 15262.508,E2 15262.508} C_VEL
LIN {X 0,Y 335.181,Z 332.261,A -85,B 0,C 180,E1 15260.772,E2 15260.772} C_VEL
LIN {X 0,Y 338.644,Z 339.138,A -85,B 0,C 180,E1 15258.584,E2 15258.584} C_VEL
LIN {X 0,Y 343.572,Z 350.049,A -85,B 0,C 180,E1 15255.581,E2 15255.581} C_VEL
LIN {X 0,Y 354.646,Z 366.45,A -85,B 0,C 180,E1 15253.096,E2 15253.096} C_VEL
LIN {X 0,Y 365.235,Z 383.822,A -85,B 0,C 180,E1 15250.924,E2 15250.924} C_VEL
LIN {X 0,Y 371.372,Z 395.131,A -85,B 0,C 180,E1 15249.731,E2 15249.731} C_VEL
LIN {X 0,Y 365.497,Z 566.215,A -85,B 0,C 180,E1 15246.469,E2 15246.469} C_VEL
LIN {X 0,Y 364.483,Z 584.95,A -85,B 0,C 180,E1 15245.856,E2 15245.856} C_VEL
LIN {X 0,Y 362.848,Z 602.649,A -85,B 0,C 180,E1 15245.023,E2 15245.023} C_VEL
LIN {X 0,Y 360.528,Z 620.805,A -85,B 0,C 180,E1 15243.878,E2 15243.878} C_VEL
LIN {X 0,Y 357.652,Z 638.242,A -85,B 0,C 180,E1 15242.462,E2 15242.462} C_VEL
LIN {X 0,Y 354.406,Z 654.561,A -85,B 0,C 180,E1 15240.8,E2 15240.8} C_VEL
LIN {X 0,Y 350.903,Z 669.814,A -85,B 0,C 180,E1 15238.879,E2 15238.879} C_VEL
LIN {X 0,Y 347.276,Z 683.981,A -85,B 0,C 180,E1 15236.688,E2 15236.688} C_VEL
LIN {X 0,Y 343.882,Z 696.2,A -85,B 0,C 180,E1 15234.385,E2 15234.385} C_VEL
LIN {X 0,Y 340.482,Z 707.778,A -85,B 0,C 180,E1 15231.716,E2 15231.716} C_VEL
LIN {X 0,Y 337.476,Z 717.82,A -85,B 0,C 180,E1 15228.84,E2 15228.84} C_VEL
LIN {X 0,Y 334.91,Z 726.341,A -85,B 0,C 180,E1 15225.764,E2 15225.764} C_VEL
LIN {X 0,Y 332.895,Z 733.313,A -85,B 0,C 180,E1 15222.489,E2 15222.489} C_VEL
LIN {X 0,Y 331.513,Z 738.445,A -85,B 0,C 180,E1 15219.198,E2 15219.198} C_VEL
LIN {X 0,Y 330.607,Z 742.054,A -85,B 0,C 180,E1 15215.728,E2 15215.728} C_VEL
LIN {X 0,Y 330.182,Z 743.952,A -85,B 0,C 180,E1 15212.256,E2 15212.256} C_VEL
LIN {X 0,Y 330.123,Z 744.22,A -85,B 0,C 180,E1 15208.785,E2 15208.785} C_VEL
LIN {X 0,Y 330.425,Z 742.87,A -85,B 0,C 180,E1 15205.314,E2 15205.314} C_VEL
LIN {X 0,Y 331.162,Z 739.844,A -85,B 0,C 180,E1 15201.842,E2 15201.842} C_VEL
LIN {X 0,Y 332.361,Z 735.3,A -85,B 0,C 180,E1 15198.548,E2 15198.548} C_VEL
LIN {X 0,Y 334.15,Z 728.997,A -85,B 0,C 180,E1 15195.266,E2 15195.266} C_VEL
LIN {X 0,Y 336.491,Z 721.192,A -85,B 0,C 180,E1 15192.179,E2 15192.179} C_VEL
LIN {X 0,Y 337.17,Z 718.967,A -85,B 0,C 180,E1 15191.419,E2 15191.419} C_VEL
LIN {X 0,Y 337.295,Z 715.6,A -85,B 0,C 180,E1 15190.238,E2 15190.238} C_VEL
LIN {X 0,Y 334.749,Z 706.748,A -85,B 0,C 180,E1 15187.184,E2 15187.184} C_VEL
LIN {X 0,Y 335.198,Z 702.513,A -85,B 0,C 180,E1 15186.068,E2 15186.068} C_VEL
LIN {X 0,Y 338.821,Z 690.407,A -85,B 0,C 180,E1 15183.539,E2 15183.539} C_VEL
LIN {X 0,Y 342.603,Z 676.785,A -85,B 0,C 180,E1 15181.215,E2 15181.215} C_VEL
LIN {X 0,Y 346.299,Z 662.101,A -85,B 0,C 180,E1 15179.171,E2 15179.171} C_VEL
LIN {X 0,Y 349.849,Z 646.05,A -85,B 0,C 180,E1 15177.358,E2 15177.358} C_VEL
LIN {X 0,Y 352.911,Z 629.764,A -85,B 0,C 180,E1 15175.878,E2 15175.878} C_VEL
LIN {X 0,Y 355.587,Z 612.062,A -85,B 0,C 180,E1 15174.604,E2 15174.604} C_VEL
LIN {X 0,Y 357.708,Z 593.156,A -85,B 0,C 180,E1 15173.573,E2 15173.573} C_VEL
LIN {X 0,Y 359.098,Z 573.733,A -85,B 0,C 180,E1 15172.823,E2 15172.823} C_VEL
LIN {X 0,Y 359.921,Z 549.235,A -85,B 0,C 180,E1 15172.243,E2 15172.243} C_VEL
LIN {X 0,Y 365.403,Z 397.808,A -85,B 0,C 180,E1 15169.34,E2 15169.34} C_VEL
LIN {X 0,Y 355.071,Z 379.673,A -85,B 0,C 180,E1 15167.215,E2 15167.215} C_VEL
LIN {X 0,Y 345.298,Z 364.445,A -85,B 0,C 180,E1 15165.06,E2 15165.06} C_VEL
LIN {X 0,Y 335.772,Z 350.784,A -85,B 0,C 180,E1 15162.761,E2 15162.761} C_VEL
LIN {X 0,Y 331.864,Z 342.522,A -85,B 0,C 180,E1 15160.339,E2 15160.339} C_VEL
LIN {X 0,Y 328.69,Z 335.771,A -85,B 0,C 180,E1 15158.135,E2 15158.135} C_VEL
LIN {X 0,Y 326.623,Z 331.539,A -85,B 0,C 180,E1 15156.651,E2 15156.651} C_VEL
LIN {X 0,Y 324.81,Z 328.032,A -85,B 0,C 180,E1 15155.341,E2 15155.341} C_VEL
LIN {X 0,Y 322.269,Z 323.301,A -85,B 0,C 180,E1 15153.43,E2 15153.43} C_VEL
LIN {X 0,Y 322.076,Z 322.376,A -85,B 0,C 180,E1 15152.907,E2 15152.907} C_VEL
LIN {X 0,Y 322.074,Z 322.345,A -85,B 0,C 180,E1 15148.535,E2 15148.535} C_VEL
LIN {X 0,Y 322.084,Z 322.337,A -85,B 0,C 180,E1 15144.126,E2 15144.126} C_VEL
LIN {X 0,Y 322.092,Z 322.332,A -85,B 0,C 180,E1 15139.778,E2 15139.778} C_VEL
LIN {X 0,Y 322.088,Z 322.339,A -85,B 0,C 180,E1 15135.484,E2 15135.484} C_VEL
LIN {X 0,Y 322.064,Z 322.365,A -85,B 0,C 180,E1 15131.098,E2 15131.098} C_VEL
LIN {X 0,Y 322.048,Z 322.354,A -85,B 0,C 180,E1 15126.776,E2 15126.776} C_VEL
LIN {X 0,Y 322.04,Z 322.336,A -85,B 0,C 180,E1 15122.314,E2 15122.314} C_VEL
LIN {X 0,Y 322.046,Z 322.337,A -85,B 0,C 180,E1 15118.043,E2 15118.043} C_VEL
LIN {X 0,Y 322.081,Z 322.351,A -85,B 0,C 180,E1 15113.584,E2 15113.584} C_VEL
LIN {X 0,Y 322.082,Z 322.365,A -85,B 0,C 180,E1 15109.266,E2 15109.266} C_VEL
LIN {X 0,Y 322.069,Z 322.351,A -85,B 0,C 180,E1 15104.884,E2 15104.884} C_VEL
LIN {X 0,Y 322.064,Z 322.345,A -85,B 0,C 180,E1 15100.599,E2 15100.599} C_VEL
LIN {X 0,Y 322.066,Z 322.345,A -85,B 0,C 180,E1 15096.198,E2 15096.198} C_VEL
LIN {X 0,Y 322.141,Z 322.707,A -85,B 0,C 180,E1 15095.522,E2 15095.522} C_VEL
LIN {X 0,Y 323.78,Z 326.39,A -85,B 0,C 180,E1 15094.188,E2 15094.188} C_VEL
LIN {X 0,Y 325.054,Z 327.877,A -85,B 0,C 180,E1 15093.512,E2 15093.512} C_VEL
LIN {X 0,Y 326.832,Z 331.6,A -85,B 0,C 180,E1 15092.29,E2 15092.29} C_VEL
LIN {X 0,Y 328.017,Z 333.531,A -85,B 0,C 180,E1 15091.607,E2 15091.607} C_VEL
LIN {X 0,Y 330.931,Z 338.973,A -85,B 0,C 180,E1 15089.898,E2 15089.898} C_VEL
LIN {X 0,Y 335.271,Z 347.087,A -85,B 0,C 180,E1 15087.534,E2 15087.534} C_VEL
LIN {X 0,Y 341.078,Z 358.854,A -85,B 0,C 180,E1 15084.52,E2 15084.52} C_VEL
LIN {X 0,Y 347.447,Z 373.012,A -85,B 0,C 180,E1 15081.357,E2 15081.357} C_VEL
LIN {X 0,Y 349.493,Z 377.491,A -85,B 0,C 180,E1 15080.519,E2 15080.519} C_VEL
LIN {X 0,Y 359.941,Z 395.515,A -85,B 0,C 180,E1 15078.242,E2 15078.242} C_VEL
LIN {X 0,Y 363.916,Z 403.32,A -85,B 0,C 180,E1 15077.407,E2 15077.407} C_VEL
LIN {X 0,Y 365.906,Z 432.308,A -85,B 0,C 180,E1 15076.299,E2 15076.299} C_VEL
LIN {X 0,Y 356.749,Z 630.067,A -85,B 0,C 180,E1 15072.06,E2 15072.06} C_VEL
LIN {X 0,Y 354.599,Z 651.963,A -85,B 0,C 180,E1 15071.331,E2 15071.331} C_VEL
LIN {X 0,Y 351.557,Z 673.11,A -85,B 0,C 180,E1 15070.341,E2 15070.341} C_VEL
LIN {X 0,Y 348.102,Z 693.035,A -85,B 0,C 180,E1 15069.084,E2 15069.084} C_VEL
LIN {X 0,Y 344.385,Z 711.851,A -85,B 0,C 180,E1 15067.566,E2 15067.566} C_VEL
LIN {X 0,Y 340.48,Z 729.939,A -85,B 0,C 180,E1 15065.758,E2 15065.758} C_VEL
LIN {X 0,Y 336.537,Z 747.239,A -85,B 0,C 180,E1 15063.647,E2 15063.647} C_VEL
LIN {X 0,Y 332.731,Z 763.666,A -85,B 0,C 180,E1 15061.221,E2 15061.221} C_VEL
LIN {X 0,Y 329.186,Z 779.091,A -85,B 0,C 180,E1 15058.48,E2 15058.48} C_VEL
LIN {X 0,Y 326.291,Z 792.623,A -85,B 0,C 180,E1 15055.598,E2 15055.598} C_VEL
LIN {X 0,Y 323.958,Z 804.798,A -85,B 0,C 180,E1 15052.501,E2 15052.501} C_VEL
LIN {X 0,Y 322.282,Z 815.558,A -85,B 0,C 180,E1 15049.199,E2 15049.199} C_VEL
LIN {X 0,Y 321.288,Z 824.772,A -85,B 0,C 180,E1 15045.708,E2 15045.708} C_VEL
LIN {X 0,Y 320.898,Z 832.016,A -85,B 0,C 180,E1 15042.232,E2 15042.232} C_VEL
LIN {X 0,Y 320.976,Z 837.44,A -85,B 0,C 180,E1 15038.78,E2 15038.78} C_VEL
LIN {X 0,Y 321.244,Z 841.106,A -85,B 0,C 180,E1 15035.358,E2 15035.358} C_VEL
LIN {X 0,Y 321.466,Z 842.897,A -85,B 0,C 180,E1 15032.317,E2 15032.317} C_VEL
LIN {X 0,Y 321.525,Z 843.248,A -85,B 0,C 180,E1 15029.287,E2 15029.287} C_VEL
LIN {X 0,Y 321.372,Z 842.247,A -85,B 0,C 180,E1 15026.254,E2 15026.254} C_VEL
LIN {X 0,Y 321.104,Z 839.572,A -85,B 0,C 180,E1 15023.025,E2 15023.025} C_VEL
LIN {X 0,Y 320.905,Z 835.086,A -85,B 0,C 180,E1 15019.589,E2 15019.589} C_VEL
LIN {X 0,Y 320.995,Z 829.211,A -85,B 0,C 180,E1 15016.307,E2 15016.307} C_VEL
LIN {X 0,Y 321.615,Z 821.111,A -85,B 0,C 180,E1 15012.822,E2 15012.822} C_VEL
LIN {X 0,Y 322.849,Z 811.545,A -85,B 0,C 180,E1 15009.516,E2 15009.516} C_VEL
LIN {X 0,Y 324.686,Z 800.665,A -85,B 0,C 180,E1 15006.402,E2 15006.402} C_VEL
LIN {X 0,Y 327.285,Z 787.743,A -85,B 0,C 180,E1 15003.316,E2 15003.316} C_VEL
LIN {X 0,Y 330.473,Z 773.361,A -85,B 0,C 180,E1 15000.452,E2 15000.452} C_VEL
LIN {X 0,Y 334.021,Z 758.021,A -85,B 0,C 180,E1 14997.901,E2 14997.901} C_VEL
LIN {X 0,Y 337.894,Z 741.294,A -85,B 0,C 180,E1 14995.586,E2 14995.586} C_VEL
LIN {X 0,Y 341.994,Z 723.02,A -85,B 0,C 180,E1 14993.513,E2 14993.513} C_VEL
LIN {X 0,Y 345.892,Z 704.249,A -85,B 0,C 180,E1 14991.787,E2 14991.787} C_VEL
LIN {X 0,Y 349.539,Z 684.748,A -85,B 0,C 180,E1 14990.367,E2 14990.367} C_VEL
LIN {X 0,Y 352.746,Z 665.005,A -85,B 0,C 180,E1 14989.26,E2 14989.26} C_VEL
LIN {X 0,Y 355.371,Z 644.534,A -85,B 0,C 180,E1 14988.409,E2 14988.409} C_VEL
LIN {X 0,Y 357.081,Z 623.395,A -85,B 0,C 180,E1 14987.788,E2 14987.788} C_VEL
LIN {X 0,Y 365.863,Z 430.43,A -85,B 0,C 180,E1 14983.668,E2 14983.668} C_VEL
LIN {X 0,Y 363.563,Z 402.371,A -85,B 0,C 180,E1 14982.547,E2 14982.547} C_VEL
LIN {X 0,Y 353.314,Z 383.877,A -85,B 0,C 180,E1 14980.368,E2 14980.368} C_VEL
LIN {X 0,Y 348.685,Z 375.951,A -85,B 0,C 180,E1 14979.267,E2 14979.267} C_VEL
LIN {X 0,Y 342.375,Z 361.611,A -85,B 0,C 180,E1 14976.15,E2 14976.15} C_VEL
LIN {X 0,Y 336.776,Z 350.046,A -85,B 0,C 180,E1 14973.315,E2 14973.315} C_VEL
LIN {X 0,Y 332.063,Z 341.072,A -85,B 0,C 180,E1 14970.789,E2 14970.789} C_VEL
LIN {X 0,Y 329.674,Z 336.622,A -85,B 0,C 180,E1 14969.427,E2 14969.427} C_VEL
LIN {X 0,Y 327.403,Z 332.26,A -85,B 0,C 180,E1 14968.048,E2 14968.048} C_VEL
LIN {X 0,Y 325.38,Z 328.95,A -85,B 0,C 180,E1 14966.853,E2 14966.853} C_VEL
LIN {X 0,Y 324.665,Z 327.308,A -85,B 0,C 180,E1 14966.325,E2 14966.325} C_VEL
LIN {X 0,Y 322.623,Z 324.406,A -85,B 0,C 180,E1 14965.124,E2 14965.124} C_VEL
LIN {X 0,Y 322.127,Z 322.599,A -85,B 0,C 180,E1 14964.48,E2 14964.48} C_VEL
LIN {X 0,Y 322.095,Z 322.363,A -85,B 0,C 180,E1 14960.535,E2 14960.535} C_VEL
LIN {X 0,Y 322.076,Z 322.366,A -85,B 0,C 180,E1 14956.224,E2 14956.224} C_VEL
LIN {X 0,Y 322.06,Z 322.349,A -85,B 0,C 180,E1 14952.005,E2 14952.005} C_VEL
LIN {X 0,Y 322.048,Z 322.338,A -85,B 0,C 180,E1 14947.672,E2 14947.672} C_VEL
LIN {X 0,Y 322.043,Z 322.338,A -85,B 0,C 180,E1 14943.381,E2 14943.381} C_VEL
LIN {X 0,Y 322.048,Z 322.359,A -85,B 0,C 180,E1 14939.11,E2 14939.11} C_VEL
LIN {X 0,Y 322.069,Z 322.364,A -85,B 0,C 180,E1 14934.656,E2 14934.656} C_VEL
LIN {X 0,Y 322.075,Z 322.336,A -85,B 0,C 180,E1 14930.349,E2 14930.349} C_VEL
LIN {X 0,Y 322.068,Z 322.333,A -85,B 0,C 180,E1 14925.986,E2 14925.986} C_VEL
LIN {X 0,Y 322.066,Z 322.347,A -85,B 0,C 180,E1 14921.726,E2 14921.726} C_VEL
LIN {X 0,Y 322.061,Z 322.365,A -85,B 0,C 180,E1 14917.358,E2 14917.358} C_VEL
LIN {X 0,Y 322.072,Z 322.368,A -85,B 0,C 180,E1 14912.847,E2 14912.847} C_VEL
LIN {X 0,Y 322.087,Z 322.36,A -85,B 0,C 180,E1 14908.565,E2 14908.565} C_VEL
LIN {X 0,Y 322.124,Z 322.658,A -85,B 0,C 180,E1 14906.674,E2 14906.674} C_VEL
LIN {X 0,Y 323.828,Z 326.438,A -85,B 0,C 180,E1 14905.165,E2 14905.165} C_VEL
LIN {X 0,Y 324.865,Z 328.259,A -85,B 0,C 180,E1 14904.429,E2 14904.429} C_VEL
LIN {X 0,Y 327.192,Z 332.729,A -85,B 0,C 180,E1 14902.766,E2 14902.766} C_VEL
LIN {X 0,Y 331.233,Z 340.957,A -85,B 0,C 180,E1 14899.987,E2 14899.987} C_VEL
LIN {X 0,Y 335.521,Z 350.368,A -85,B 0,C 180,E1 14897.199,E2 14897.199} C_VEL
LIN {X 0,Y 344.557,Z 363.411,A -85,B 0,C 180,E1 14894.981,E2 14894.981} C_VEL
LIN {X 0,Y 353.664,Z 377.534,A -85,B 0,C 180,E1 14892.956,E2 14892.956} C_VEL
LIN {X 0,Y 364.235,Z 395.671,A -85,B 0,C 180,E1 14890.776,E2 14890.776} C_VEL
LIN {X 0,Y 365.435,Z 398.292,A -85,B 0,C 180,E1 14890.528,E2 14890.528} C_VEL
LIN {X 0,Y 359.336,Z 566.906,A -85,B 0,C 180,E1 14887.269,E2 14887.269} C_VEL
LIN {X 0,Y 358.271,Z 585.725,A -85,B 0,C 180,E1 14886.646,E2 14886.646} C_VEL
LIN {X 0,Y 356.526,Z 603.807,A -85,B 0,C 180,E1 14885.782,E2 14885.782} C_VEL
LIN {X 0,Y 354.199,Z 621.302,A -85,B 0,C 180,E1 14884.666,E2 14884.666} C_VEL
LIN {X 0,Y 351.205,Z 638.841,A -85,B 0,C 180,E1 14883.231,E2 14883.231} C_VEL
LIN {X 0,Y 347.815,Z 655.243,A -85,B 0,C 180,E1 14881.546,E2 14881.546} C_VEL
LIN {X 0,Y 344.163,Z 670.564,A -85,B 0,C 180,E1 14879.595,E2 14879.595} C_VEL
LIN {X 0,Y 340.5,Z 684.31,A -85,B 0,C 180,E1 14877.452,E2 14877.452} C_VEL
LIN {X 0,Y 336.691,Z 697.465,A -85,B 0,C 180,E1 14874.941,E2 14874.941} C_VEL
LIN {X 0,Y 333.135,Z 709.024,A -85,B 0,C 180,E1 14872.22,E2 14872.22} C_VEL
LIN {X 0,Y 329.981,Z 719.051,A -85,B 0,C 180,E1 14869.285,E2 14869.285} C_VEL
LIN {X 0,Y 327.283,Z 727.563,A -85,B 0,C 180,E1 14866.141,E2 14866.141} C_VEL
LIN {X 0,Y 325.156,Z 734.527,A -85,B 0,C 180,E1 14862.791,E2 14862.791} C_VEL
LIN {X 0,Y 323.692,Z 739.654,A -85,B 0,C 180,E1 14859.422,E2 14859.422} C_VEL
LIN {X 0,Y 322.732,Z 743.258,A -85,B 0,C 180,E1 14855.868,E2 14855.868} C_VEL
LIN {X 0,Y 322.279,Z 745.154,A -85,B 0,C 180,E1 14852.311,E2 14852.311} C_VEL
LIN {X 0,Y 322.215,Z 745.422,A -85,B 0,C 180,E1 14848.755,E2 14848.755} C_VEL
LIN {X 0,Y 322.536,Z 744.073,A -85,B 0,C 180,E1 14845.199,E2 14845.199} C_VEL
LIN {X 0,Y 323.32,Z 741.048,A -85,B 0,C 180,E1 14841.643,E2 14841.643} C_VEL
LIN {X 0,Y 324.591,Z 736.51,A -85,B 0,C 180,E1 14838.27,E2 14838.27} C_VEL
LIN {X 0,Y 326.483,Z 730.211,A -85,B 0,C 180,E1 14834.912,E2 14834.912} C_VEL
LIN {X 0,Y 328.949,Z 722.415,A -85,B 0,C 180,E1 14831.756,E2 14831.756} C_VEL
LIN {X 0,Y 331.87,Z 713.174,A -85,B 0,C 180,E1 14828.806,E2 14828.806} C_VEL
LIN {X 0,Y 335.198,Z 702.513,A -85,B 0,C 180,E1 14826.068,E2 14826.068} C_VEL
LIN {X 0,Y 335.725,Z 698.146,A -85,B 0,C 180,E1 14824.973,E2 14824.973} C_VEL
LIN {X 0,Y 334.106,Z 687.632,A -85,B 0,C 180,E1 14822.275,E2 14822.275} C_VEL
LIN {X 0,Y 334.506,Z 682.533,A -85,B 0,C 180,E1 14821.275,E2 14821.275} C_VEL
LIN {X 0,Y 334.7,Z 681.744,A -85,B 0,C 180,E1 14821.146,E2 14821.146} C_VEL
LIN {X 0,Y 338.614,Z 667.296,A -85,B 0,C 180,E1 14818.986,E2 14818.986} C_VEL
LIN {X 0,Y 342.34,Z 651.752,A -85,B 0,C 180,E1 14817.096,E2 14817.096} C_VEL
LIN {X 0,Y 345.87,Z 634.511,A -85,B 0,C 180,E1 14815.417,E2 14815.417} C_VEL
LIN {X 0,Y 348.705,Z 617.506,A -85,B 0,C 180,E1 14814.101,E2 14814.101} C_VEL
LIN {X 0,Y 351.098,Z 598.691,A -85,B 0,C 180,E1 14812.985,E2 14812.985} C_VEL
LIN {X 0,Y 352.734,Z 579.403,A -85,B 0,C 180,E1 14812.157,E2 14812.157} C_VEL
LIN {X 0,Y 353.592,Z 559.428,A -85,B 0,C 180,E1 14811.603,E2 14811.603} C_VEL
LIN {X 0,Y 359.51,Z 400.832,A -85,B 0,C 180,E1 14808.507,E2 14808.507} C_VEL
LIN {X 0,Y 349.361,Z 383.174,A -85,B 0,C 180,E1 14806.333,E2 14806.333} C_VEL
LIN {X 0,Y 340.387,Z 369.124,A -85,B 0,C 180,E1 14804.268,E2 14804.268} C_VEL
LIN {X 0,Y 331.339,Z 356.057,A -85,B 0,C 180,E1 14802.003,E2 14802.003} C_VEL
LIN {X 0,Y 327.737,Z 351.036,A -85,B 0,C 180,E1 14800.99,E2 14800.99} C_VEL
LIN {X 0,Y 323.667,Z 342.153,A -85,B 0,C 180,E1 14798.159,E2 14798.159} C_VEL
LIN {X 0,Y 320.744,Z 336.628,A -85,B 0,C 180,E1 14796.099,E2 14796.099} C_VEL
LIN {X 0,Y 318.81,Z 332.641,A -85,B 0,C 180,E1 14794.587,E2 14794.587} C_VEL
LIN {X 0,Y 316.469,Z 328.067,A -85,B 0,C 180,E1 14792.702,E2 14792.702} C_VEL
LIN {X 0,Y 314.358,Z 324.467,A -85,B 0,C 180,E1 14791.016,E2 14791.016} C_VEL
LIN {X 0,Y 314.145,Z 323.364,A -85,B 0,C 180,E1 14790.4,E2 14790.4} C_VEL
LIN {X 0,Y 314.152,Z 323.333,A -85,B 0,C 180,E1 14786.054,E2 14786.054} C_VEL
LIN {X 0,Y 314.166,Z 323.343,A -85,B 0,C 180,E1 14781.665,E2 14781.665} C_VEL
LIN {X 0,Y 314.136,Z 323.353,A -85,B 0,C 180,E1 14777.218,E2 14777.218} C_VEL
LIN {X 0,Y 314.117,Z 323.332,A -85,B 0,C 180,E1 14772.875,E2 14772.875} C_VEL
LIN {X 0,Y 314.108,Z 323.321,A -85,B 0,C 180,E1 14768.42,E2 14768.42} C_VEL
LIN {X 0,Y 314.115,Z 323.328,A -85,B 0,C 180,E1 14764.016,E2 14764.016} C_VEL
LIN {X 0,Y 314.135,Z 323.35,A -85,B 0,C 180,E1 14759.636,E2 14759.636} C_VEL
LIN {X 0,Y 314.13,Z 323.341,A -85,B 0,C 180,E1 14755.253,E2 14755.253} C_VEL
LIN {X 0,Y 314.119,Z 323.327,A -85,B 0,C 180,E1 14750.843,E2 14750.843} C_VEL
LIN {X 0,Y 314.115,Z 323.325,A -85,B 0,C 180,E1 14746.376,E2 14746.376} C_VEL
LIN {X 0,Y 314.123,Z 323.329,A -85,B 0,C 180,E1 14742.016,E2 14742.016} C_VEL
LIN {X 0,Y 314.163,Z 323.599,A -85,B 0,C 180,E1 14738.139,E2 14738.139} C_VEL
LIN {X 0,Y 315.937,Z 327.481,A -85,B 0,C 180,E1 14736.5,E2 14736.5} C_VEL
LIN {X 0,Y 317.329,Z 329.355,A -85,B 0,C 180,E1 14735.622,E2 14735.622} C_VEL
LIN {X 0,Y 319.354,Z 333.115,A -85,B 0,C 180,E1 14734.203,E2 14734.203} C_VEL
LIN {X 0,Y 320.252,Z 334.58,A -85,B 0,C 180,E1 14733.639,E2 14733.639} C_VEL
LIN {X 0,Y 322.938,Z 339.463,A -85,B 0,C 180,E1 14731.926,E2 14731.926} C_VEL
LIN {X 0,Y 327.639,Z 348.178,A -85,B 0,C 180,E1 14729.157,E2 14729.157} C_VEL
LIN {X 0,Y 333.815,Z 360.651,A -85,B 0,C 180,E1 14725.729,E2 14725.729} C_VEL
LIN {X 0,Y 340.38,Z 375.126,A -85,B 0,C 180,E1 14722.339,E2 14722.339} C_VEL
LIN {X 0,Y 349.582,Z 390.621,A -85,B 0,C 180,E1 14720.105,E2 14720.105} C_VEL
LIN {X 0,Y 358.311,Z 406.665,A -85,B 0,C 180,E1 14718.184,E2 14718.184} C_VEL
LIN {X 0,Y 360.026,Z 433.456,A -85,B 0,C 180,E1 14717.144,E2 14717.144} C_VEL
LIN {X 0,Y 350.599,Z 629.113,A -85,B 0,C 180,E1 14712.904,E2 14712.904} C_VEL
LIN {X 0,Y 348.388,Z 650.993,A -85,B 0,C 180,E1 14712.168,E2 14712.168} C_VEL
LIN {X 0,Y 345.208,Z 672.311,A -85,B 0,C 180,E1 14711.162,E2 14711.162} C_VEL
LIN {X 0,Y 341.563,Z 692.518,A -85,B 0,C 180,E1 14709.871,E2 14709.871} C_VEL
LIN {X 0,Y 337.601,Z 711.697,A -85,B 0,C 180,E1 14708.295,E2 14708.295} C_VEL
LIN {X 0,Y 333.449,Z 730.002,A -85,B 0,C 180,E1 14706.419,E2 14706.419} C_VEL
LIN {X 0,Y 329.348,Z 747.107,A -85,B 0,C 180,E1 14704.273,E2 14704.273} C_VEL
LIN {X 0,Y 325.365,Z 763.368,A -85,B 0,C 180,E1 14701.804,E2 14701.804} C_VEL
LIN {X 0,Y 321.656,Z 778.655,A -85,B 0,C 180,E1 14699.006,E2 14699.006} C_VEL
LIN {X 0,Y 318.447,Z 792.826,A -85,B 0,C 180,E1 14695.876,E2 14695.876} C_VEL
LIN {X 0,Y 315.919,Z 805.393,A -85,B 0,C 180,E1 14692.516,E2 14692.516} C_VEL
LIN {X 0,Y 314.217,Z 815.959,A -85,B 0,C 180,E1 14689.079,E2 14689.079} C_VEL
LIN {X 0,Y 313.267,Z 824.77,A -85,B 0,C 180,E1 14685.551,E2 14685.551} C_VEL
LIN {X 0,Y 312.918,Z 831.796,A -85,B 0,C 180,E1 14681.987,E2 14681.987} C_VEL
LIN {X 0,Y 313.033,Z 836.689,A -85,B 0,C 180,E1 14678.634,E2 14678.634} C_VEL
LIN {X 0,Y 313.346,Z 840.164,A -85,B 0,C 180,E1 14675.126,E2 14675.126} C_VEL
LIN {X 0,Y 313.56,Z 841.841,A -85,B 0,C 180,E1 14672.01,E2 14672.01} C_VEL
LIN {X 0,Y 313.609,Z 841.993,A -85,B 0,C 180,E1 14668.904,E2 14668.904} C_VEL
LIN {X 0,Y 313.402,Z 840.687,A -85,B 0,C 180,E1 14665.609,E2 14665.609} C_VEL
LIN {X 0,Y 313.116,Z 837.976,A -85,B 0,C 180,E1 14662.477,E2 14662.477} C_VEL
LIN {X 0,Y 312.929,Z 833.554,A -85,B 0,C 180,E1 14659.134,E2 14659.134} C_VEL
LIN {X 0,Y 313.098,Z 827.154,A -85,B 0,C 180,E1 14655.577,E2 14655.577} C_VEL
LIN {X 0,Y 313.791,Z 819.369,A -85,B 0,C 180,E1 14652.189,E2 14652.189} C_VEL
LIN {X 0,Y 315.279,Z 809.11,A -85,B 0,C 180,E1 14648.611,E2 14648.611} C_VEL
LIN {X 0,Y 317.501,Z 797.265,A -85,B 0,C 180,E1 14645.24,E2 14645.24} C_VEL
LIN {X 0,Y 320.421,Z 783.905,A -85,B 0,C 180,E1 14642.092,E2 14642.092} C_VEL
LIN {X 0,Y 323.84,Z 769.519,A -85,B 0,C 180,E1 14639.272,E2 14639.272} C_VEL
LIN {X 0,Y 327.687,Z 753.709,A -85,B 0,C 180,E1 14636.687,E2 14636.687} C_VEL
LIN {X 0,Y 331.911,Z 736.35,A -85,B 0,C 180,E1 14634.346,E2 14634.346} C_VEL
LIN {X 0,Y 336.156,Z 717.963,A -85,B 0,C 180,E1 14632.322,E2 14632.322} C_VEL
LIN {X 0,Y 340.279,Z 698.531,A -85,B 0,C 180,E1 14630.604,E2 14630.604} C_VEL
LIN {X 0,Y 343.957,Z 679.227,A -85,B 0,C 180,E1 14629.263,E2 14629.263} C_VEL
LIN {X 0,Y 347.131,Z 659.587,A -85,B 0,C 180,E1 14628.215,E2 14628.215} C_VEL
LIN {X 0,Y 349.692,Z 638.776,A -85,B 0,C 180,E1 14627.402,E2 14627.402} C_VEL
LIN {X 0,Y 351.251,Z 616.882,A -85,B 0,C 180,E1 14626.811,E2 14626.811} C_VEL
LIN {X 0,Y 359.974,Z 431.314,A -85,B 0,C 180,E1 14622.814,E2 14622.814} C_VEL
LIN {X 0,Y 357.988,Z 406.017,A -85,B 0,C 180,E1 14621.783,E2 14621.783} C_VEL
LIN {X 0,Y 347.786,Z 387.628,A -85,B 0,C 180,E1 14619.526,E2 14619.526} C_VEL
LIN {X 0,Y 340.491,Z 375.448,A -85,B 0,C 180,E1 14617.753,E2 14617.753} C_VEL
LIN {X 0,Y 334.422,Z 361.978,A -85,B 0,C 180,E1 14614.615,E2 14614.615} C_VEL
LIN {X 0,Y 328.952,Z 350.955,A -85,B 0,C 180,E1 14611.675,E2 14611.675} C_VEL
LIN {X 0,Y 324.536,Z 342.536,A -85,B 0,C 180,E1 14609.129,E2 14609.129} C_VEL
LIN {X 0,Y 321.981,Z 337.849,A -85,B 0,C 180,E1 14607.561,E2 14607.561} C_VEL
LIN {X 0,Y 319.574,Z 333.347,A -85,B 0,C 180,E1 14605.977,E2 14605.977} C_VEL
LIN {X 0,Y 317.442,Z 329.736,A -85,B 0,C 180,E1 14604.567,E2 14604.567} C_VEL
LIN {X 0,Y 316.736,Z 328.313,A -85,B 0,C 180,E1 14604.03,E2 14604.03} C_VEL
LIN {X 0,Y 314.637,Z 325.217,A -85,B 0,C 180,E1 14602.613,E2 14602.613} C_VEL
LIN {X 0,Y 314.147,Z 323.494,A -85,B 0,C 180,E1 14601.862,E2 14601.862} C_VEL
LIN {X 0,Y 314.123,Z 323.334,A -85,B 0,C 180,E1 14597.409,E2 14597.409} C_VEL
LIN {X 0,Y 314.129,Z 323.324,A -85,B 0,C 180,E1 14593.061,E2 14593.061} C_VEL
LIN {X 0,Y 314.146,Z 323.32,A -85,B 0,C 180,E1 14588.603,E2 14588.603} C_VEL
LIN {X 0,Y 314.126,Z 323.334,A -85,B 0,C 180,E1 14584.198,E2 14584.198} C_VEL
LIN {X 0,Y 314.109,Z 323.359,A -85,B 0,C 180,E1 14579.817,E2 14579.817} C_VEL
LIN {X 0,Y 314.103,Z 323.341,A -85,B 0,C 180,E1 14575.252,E2 14575.252} C_VEL
LIN {X 0,Y 314.117,Z 323.322,A -85,B 0,C 180,E1 14570.842,E2 14570.842} C_VEL
LIN {X 0,Y 314.146,Z 323.321,A -85,B 0,C 180,E1 14566.377,E2 14566.377} C_VEL
LIN {X 0,Y 314.139,Z 323.338,A -85,B 0,C 180,E1 14562.016,E2 14562.016} C_VEL
LIN {X 0,Y 314.126,Z 323.357,A -85,B 0,C 180,E1 14557.545,E2 14557.545} C_VEL
LIN {X 0,Y 314.129,Z 323.353,A -85,B 0,C 180,E1 14553.025,E2 14553.025} C_VEL
LIN {X 0,Y 314.161,Z 323.566,A -85,B 0,C 180,E1 14549.236,E2 14549.236} C_VEL
LIN {X 0,Y 315.946,Z 327.496,A -85,B 0,C 180,E1 14547.453,E2 14547.453} C_VEL
LIN {X 0,Y 316.972,Z 329.07,A -85,B 0,C 180,E1 14546.709,E2 14546.709} C_VEL
LIN {X 0,Y 318.886,Z 332.744,A -85,B 0,C 180,E1 14545.204,E2 14545.204} C_VEL
LIN {X 0,Y 321.869,Z 338.724,A -85,B 0,C 180,E1 14542.94,E2 14542.94} C_VEL
LIN {X 0,Y 325.849,Z 347.05,A -85,B 0,C 180,E1 14540.094,E2 14540.094} C_VEL
LIN {X 0,Y 328.116,Z 351.759,A -85,B 0,C 180,E1 14538.72,E2 14538.72} C_VEL
LIN {X 0,Y 337.734,Z 365.253,A -85,B 0,C 180,E1 14536.243,E2 14536.243} C_VEL
LIN {X 0,Y 347.005,Z 379.436,A -85,B 0,C 180,E1 14534.065,E2 14534.065} C_VEL
LIN {X 0,Y 356.673,Z 395.808,A -85,B 0,C 180,E1 14531.963,E2 14531.963} C_VEL
LIN {X 0,Y 359.573,Z 401.36,A -85,B 0,C 180,E1 14531.353,E2 14531.353} C_VEL
LIN {X 0,Y 353.247,Z 567.573,A -85,B 0,C 180,E1 14528.096,E2 14528.096} C_VEL
LIN {X 0,Y 352.129,Z 586.495,A -85,B 0,C 180,E1 14527.463,E2 14527.463} C_VEL
LIN {X 0,Y 350.278,Z 604.889,A -85,B 0,C 180,E1 14526.574,E2 14526.574} C_VEL
LIN {X 0,Y 347.767,Z 622.902,A -85,B 0,C 180,E1 14525.402,E2 14525.402} C_VEL
LIN {X 0,Y 344.698,Z 640.071,A -85,B 0,C 180,E1 14523.97,E2 14523.97} C_VEL
LIN {X 0,Y 341.125,Z 656.631,A -85,B 0,C 180,E1 14522.238,E2 14522.238} C_VEL
LIN {X 0,Y 337.325,Z 671.894,A -85,B 0,C 180,E1 14520.257,E2 14520.257} C_VEL
LIN {X 0,Y 333.507,Z 685.601,A -85,B 0,C 180,E1 14518.078,E2 14518.078} C_VEL
LIN {X 0,Y 329.534,Z 698.729,A -85,B 0,C 180,E1 14515.521,E2 14515.521} C_VEL
LIN {X 0,Y 325.815,Z 710.269,A -85,B 0,C 180,E1 14512.747,E2 14512.747} C_VEL
LIN {X 0,Y 322.507,Z 720.282,A -85,B 0,C 180,E1 14509.75,E2 14509.75} C_VEL
LIN {X 0,Y 319.671,Z 728.784,A -85,B 0,C 180,E1 14506.536,E2 14506.536} C_VEL
LIN {X 0,Y 317.426,Z 735.742,A -85,B 0,C 180,E1 14503.108,E2 14503.108} C_VEL
LIN {X 0,Y 315.876,Z 740.862,A -85,B 0,C 180,E1 14499.658,E2 14499.658} C_VEL
LIN {X 0,Y 314.856,Z 744.463,A -85,B 0,C 180,E1 14496.015,E2 14496.015} C_VEL
LIN {X 0,Y 314.374,Z 746.356,A -85,B 0,C 180,E1 14492.37,E2 14492.37} C_VEL
LIN {X 0,Y 314.307,Z 746.623,A -85,B 0,C 180,E1 14488.724,E2 14488.724} C_VEL
LIN {X 0,Y 314.648,Z 745.275,A -85,B 0,C 180,E1 14485.078,E2 14485.078} C_VEL
LIN {X 0,Y 315.483,Z 742.253,A -85,B 0,C 180,E1 14481.434,E2 14481.434} C_VEL
LIN {X 0,Y 316.827,Z 737.719,A -85,B 0,C 180,E1 14477.978,E2 14477.978} C_VEL
LIN {X 0,Y 318.828,Z 731.426,A -85,B 0,C 180,E1 14474.541,E2 14474.541} C_VEL
LIN {X 0,Y 321.426,Z 723.636,A -85,B 0,C 180,E1 14471.313,E2 14471.313} C_VEL
LIN {X 0,Y 324.492,Z 714.406,A -85,B 0,C 180,E1 14468.3,E2 14468.3} C_VEL
LIN {X 0,Y 327.978,Z 703.757,A -85,B 0,C 180,E1 14465.506,E2 14465.506} C_VEL
LIN {X 0,Y 331.759,Z 691.677,A -85,B 0,C 180,E1 14462.93,E2 14462.93} C_VEL
LIN {X 0,Y 334.7,Z 681.744,A -85,B 0,C 180,E1 14461.146,E2 14461.146} C_VEL
LIN {X 0,Y 335.348,Z 676.459,A -85,B 0,C 180,E1 14460.196,E2 14460.196} C_VEL
LIN {X 0,Y 334.122,Z 662.932,A -85,B 0,C 180,E1 14457.647,E2 14457.647} C_VEL
LIN {X 0,Y 334.618,Z 657.839,A -85,B 0,C 180,E1 14456.915,E2 14456.915} C_VEL
LIN {X 0,Y 334.817,Z 656.929,A -85,B 0,C 180,E1 14456.806,E2 14456.806} C_VEL
LIN {X 0,Y 338.568,Z 640.144,A -85,B 0,C 180,E1 14455.047,E2 14455.047} C_VEL
LIN {X 0,Y 341.814,Z 622.425,A -85,B 0,C 180,E1 14453.574,E2 14453.574} C_VEL
LIN {X 0,Y 344.345,Z 604.663,A -85,B 0,C 180,E1 14452.429,E2 14452.429} C_VEL
LIN {X 0,Y 346.287,Z 585.434,A -85,B 0,C 180,E1 14451.512,E2 14451.512} C_VEL
LIN {X 0,Y 347.4,Z 565.875,A -85,B 0,C 180,E1 14450.882,E2 14450.882} C_VEL
LIN {X 0,Y 353.769,Z 404.135,A -85,B 0,C 180,E1 14447.665,E2 14447.665} C_VEL
LIN {X 0,Y 343.89,Z 386.845,A -85,B 0,C 180,E1 14445.456,E2 14445.456} C_VEL
LIN {X 0,Y 334.213,Z 371.796,A -85,B 0,C 180,E1 14443.118,E2 14443.118} C_VEL
LIN {X 0,Y 325.345,Z 359.227,A -85,B 0,C 180,E1 14440.773,E2 14440.773} C_VEL
LIN {X 0,Y 319.968,Z 351.562,A -85,B 0,C 180,E1 14439.141,E2 14439.141} C_VEL
LIN {X 0,Y 315.753,Z 342.965,A -85,B 0,C 180,E1 14436.086,E2 14436.086} C_VEL
LIN {X 0,Y 313.3,Z 338.207,A -85,B 0,C 180,E1 14434.173,E2 14434.173} C_VEL
LIN {X 0,Y 311.037,Z 333.783,A -85,B 0,C 180,E1 14432.284,E2 14432.284} C_VEL
LIN {X 0,Y 309.082,Z 329.888,A -85,B 0,C 180,E1 14430.524,E2 14430.524} C_VEL
LIN {X 0,Y 306.478,Z 325.607,A -85,B 0,C 180,E1 14428.233,E2 14428.233} C_VEL
LIN {X 0,Y 306.221,Z 324.381,A -85,B 0,C 180,E1 14427.465,E2 14427.465} C_VEL
LIN {X 0,Y 306.189,Z 324.333,A -85,B 0,C 180,E1 14422.868,E2 14422.868} C_VEL
LIN {X 0,Y 306.19,Z 324.32,A -85,B 0,C 180,E1 14418.27,E2 14418.27} C_VEL
LIN {X 0,Y 306.21,Z 324.306,A -85,B 0,C 180,E1 14413.79,E2 14413.79} C_VEL
LIN {X 0,Y 306.195,Z 324.309,A -85,B 0,C 180,E1 14409.397,E2 14409.397} C_VEL
LIN {X 0,Y 306.18,Z 324.335,A -85,B 0,C 180,E1 14405.059,E2 14405.059} C_VEL
LIN {X 0,Y 306.163,Z 324.34,A -85,B 0,C 180,E1 14400.562,E2 14400.562} C_VEL
LIN {X 0,Y 306.17,Z 324.316,A -85,B 0,C 180,E1 14396.068,E2 14396.068} C_VEL
LIN {X 0,Y 306.194,Z 324.308,A -85,B 0,C 180,E1 14391.65,E2 14391.65} C_VEL
LIN {X 0,Y 306.201,Z 324.313,A -85,B 0,C 180,E1 14387.171,E2 14387.171} C_VEL
LIN {X 0,Y 306.187,Z 324.323,A -85,B 0,C 180,E1 14382.713,E2 14382.713} C_VEL
LIN {X 0,Y 306.245,Z 324.599,A -85,B 0,C 180,E1 14381.043,E2 14381.043} C_VEL
LIN {X 0,Y 307.653,Z 328.013,A -85,B 0,C 180,E1 14379.452,E2 14379.452} C_VEL
LIN {X 0,Y 309.466,Z 330.31,A -85,B 0,C 180,E1 14378.189,E2 14378.189} C_VEL
LIN {X 0,Y 311.515,Z 334.176,A -85,B 0,C 180,E1 14376.547,E2 14376.547} C_VEL
LIN {X 0,Y 312.362,Z 335.256,A -85,B 0,C 180,E1 14376.014,E2 14376.014} C_VEL
LIN {X 0,Y 314.296,Z 339.102,A -85,B 0,C 180,E1 14374.566,E2 14374.566} C_VEL
LIN {X 0,Y 315.38,Z 340.943,A -85,B 0,C 180,E1 14373.853,E2 14373.853} C_VEL
LIN {X 0,Y 318.179,Z 346.187,A -85,B 0,C 180,E1 14372.006,E2 14372.006} C_VEL
LIN {X 0,Y 322.463,Z 354.115,A -85,B 0,C 180,E1 14369.436,E2 14369.436} C_VEL
LIN {X 0,Y 328.196,Z 365.889,A -85,B 0,C 180,E1 14366.116,E2 14366.116} C_VEL
LIN {X 0,Y 332.812,Z 375.834,A -85,B 0,C 180,E1 14363.766,E2 14363.766} C_VEL
LIN {X 0,Y 342.739,Z 392.012,A -85,B 0,C 180,E1 14361.29,E2 14361.29} C_VEL
LIN {X 0,Y 351.771,Z 408.3,A -85,B 0,C 180,E1 14359.203,E2 14359.203} C_VEL
LIN {X 0,Y 352.815,Z 410.645,A -85,B 0,C 180,E1 14358.96,E2 14358.96} C_VEL
LIN {X 0,Y 354.231,Z 434.514,A -85,B 0,C 180,E1 14358.018,E2 14358.018} C_VEL
LIN {X 0,Y 344.514,Z 628.34,A -85,B 0,C 180,E1 14353.773,E2 14353.773} C_VEL
LIN {X 0,Y 342.227,Z 650.22,A -85,B 0,C 180,E1 14353.028,E2 14353.028} C_VEL
LIN {X 0,Y 338.992,Z 671.21,A -85,B 0,C 180,E1 14352.03,E2 14352.03} C_VEL
LIN {X 0,Y 335.114,Z 691.878,A -85,B 0,C 180,E1 14350.697,E2 14350.697} C_VEL
LIN {X 0,Y 330.856,Z 711.634,A -85,B 0,C 180,E1 14349.044,E2 14349.044} C_VEL
LIN {X 0,Y 326.287,Z 730.828,A -85,B 0,C 180,E1 14347.022,E2 14347.022} C_VEL
LIN {X 0,Y 321.717,Z 748.888,A -85,B 0,C 180,E1 14344.661,E2 14344.661} C_VEL
LIN {X 0,Y 317.37,Z 765.761,A -85,B 0,C 180,E1 14341.955,E2 14341.955} C_VEL
LIN {X 0,Y 313.494,Z 780.943,A -85,B 0,C 180,E1 14338.998,E2 14338.998} C_VEL
LIN {X 0,Y 310.269,Z 794.552,A -85,B 0,C 180,E1 14335.787,E2 14335.787} C_VEL
LIN {X 0,Y 307.763,Z 806.618,A -85,B 0,C 180,E1 14332.34,E2 14332.34} C_VEL
LIN {X 0,Y 306.12,Z 816.586,A -85,B 0,C 180,E1 14328.865,E2 14328.865} C_VEL
LIN {X 0,Y 305.216,Z 825.111,A -85,B 0,C 180,E1 14325.193,E2 14325.193} C_VEL
LIN {X 0,Y 304.956,Z 831.973,A -85,B 0,C 180,E1 14321.384,E2 14321.384} C_VEL
LIN {X 0,Y 305.136,Z 836.575,A -85,B 0,C 180,E1 14317.91,E2 14317.91} C_VEL
LIN {X 0,Y 305.456,Z 839.353,A -85,B 0,C 180,E1 14314.694,E2 14314.694} C_VEL
LIN {X 0,Y 305.688,Z 840.764,A -85,B 0,C 180,E1 14311.312,E2 14311.312} C_VEL
LIN {X 0,Y 305.669,Z 840.705,A -85,B 0,C 180,E1 14308.313,E2 14308.313} C_VEL
LIN {X 0,Y 305.426,Z 839.078,A -85,B 0,C 180,E1 14304.929,E2 14304.929} C_VEL
LIN {X 0,Y 305.094,Z 835.924,A -85,B 0,C 180,E1 14301.52,E2 14301.52} C_VEL
LIN {X 0,Y 304.952,Z 831.137,A -85,B 0,C 180,E1 14298.079,E2 14298.079} C_VEL
LIN {X 0,Y 305.247,Z 824.691,A -85,B 0,C 180,E1 14294.614,E2 14294.614} C_VEL
LIN {X 0,Y 306.194,Z 816.044,A -85,B 0,C 180,E1 14290.941,E2 14290.941} C_VEL
LIN {X 0,Y 307.879,Z 805.943,A -85,B 0,C 180,E1 14287.468,E2 14287.468} C_VEL
LIN {X 0,Y 310.267,Z 794.497,A -85,B 0,C 180,E1 14284.212,E2 14284.212} C_VEL
LIN {X 0,Y 313.489,Z 780.874,A -85,B 0,C 180,E1 14281.002,E2 14281.002} C_VEL
LIN {X 0,Y 317.364,Z 765.673,A -85,B 0,C 180,E1 14278.044,E2 14278.044} C_VEL
LIN {X 0,Y 321.709,Z 748.778,A -85,B 0,C 180,E1 14275.338,E2 14275.338} C_VEL
LIN {X 0,Y 326.277,Z 730.691,A -85,B 0,C 180,E1 14272.976,E2 14272.976} C_VEL
LIN {X 0,Y 330.824,Z 711.548,A -85,B 0,C 180,E1 14270.962,E2 14270.962} C_VEL
LIN {X 0,Y 334.859,Z 692.812,A -85,B 0,C 180,E1 14269.39,E2 14269.39} C_VEL
LIN {X 0,Y 338.64,Z 672.793,A -85,B 0,C 180,E1 14268.077,E2 14268.077} C_VEL
LIN {X 0,Y 341.824,Z 652.571,A -85,B 0,C 180,E1 14267.087,E2 14267.087} C_VEL
LIN {X 0,Y 344.13,Z 631.847,A -85,B 0,C 180,E1 14266.348,E2 14266.348} C_VEL
LIN {X 0,Y 345.878,Z 601.735,A -85,B 0,C 180,E1 14265.624,E2 14265.624} C_VEL
LIN {X 0,Y 354.16,Z 432.103,A -85,B 0,C 180,E1 14261.929,E2 14261.929} C_VEL
LIN {X 0,Y 352.517,Z 409.813,A -85,B 0,C 180,E1 14261.006,E2 14261.006} C_VEL
LIN {X 0,Y 342.98,Z 392.513,A -85,B 0,C 180,E1 14258.812,E2 14258.812} C_VEL
LIN {X 0,Y 332.766,Z 375.811,A -85,B 0,C 180,E1 14256.266,E2 14256.266} C_VEL
LIN {X 0,Y 327.862,Z 365.182,A -85,B 0,C 180,E1 14253.713,E2 14253.713} C_VEL
LIN {X 0,Y 322.081,Z 353.383,A -85,B 0,C 180,E1 14250.398,E2 14250.398} C_VEL
LIN {X 0,Y 317.199,Z 344.202,A -85,B 0,C 180,E1 14247.4,E2 14247.4} C_VEL
LIN {X 0,Y 314.49,Z 339.342,A -85,B 0,C 180,E1 14245.619,E2 14245.619} C_VEL
LIN {X 0,Y 312.477,Z 335.635,A -85,B 0,C 180,E1 14244.178,E2 14244.178} C_VEL
LIN {X 0,Y 309.559,Z 330.605,A -85,B 0,C 180,E1 14242.004,E2 14242.004} C_VEL
LIN {X 0,Y 308.589,Z 329.111,A -85,B 0,C 180,E1 14241.277,E2 14241.277} C_VEL
LIN {X 0,Y 306.537,Z 325.874,A -85,B 0,C 180,E1 14239.631,E2 14239.631} C_VEL
LIN {X 0,Y 306.22,Z 324.376,A -85,B 0,C 180,E1 14238.81,E2 14238.81} C_VEL
LIN {X 0,Y 306.203,Z 324.314,A -85,B 0,C 180,E1 14234.369,E2 14234.369} C_VEL
LIN {X 0,Y 306.182,Z 324.327,A -85,B 0,C 180,E1 14229.966,E2 14229.966} C_VEL
LIN {X 0,Y 306.172,Z 324.348,A -85,B 0,C 180,E1 14225.434,E2 14225.434} C_VEL
LIN {X 0,Y 306.18,Z 324.328,A -85,B 0,C 180,E1 14220.935,E2 14220.935} C_VEL
LIN {X 0,Y 306.186,Z 324.31,A -85,B 0,C 180,E1 14216.442,E2 14216.442} C_VEL
LIN {X 0,Y 306.188,Z 324.311,A -85,B 0,C 180,E1 14212.117,E2 14212.117} C_VEL
LIN {X 0,Y 306.171,Z 324.33,A -85,B 0,C 180,E1 14207.53,E2 14207.53} C_VEL
LIN {X 0,Y 306.179,Z 324.346,A -85,B 0,C 180,E1 14203.096,E2 14203.096} C_VEL
LIN {X 0,Y 306.205,Z 324.327,A -85,B 0,C 180,E1 14198.527,E2 14198.527} C_VEL
LIN {X 0,Y 306.212,Z 324.318,A -85,B 0,C 180,E1 14194.052,E2 14194.052} C_VEL
LIN {X 0,Y 306.262,Z 324.613,A -85,B 0,C 180,E1 14192.063,E2 14192.063} C_VEL
LIN {X 0,Y 307.646,Z 327.976,A -85,B 0,C 180,E1 14190.395,E2 14190.395} C_VEL
LIN {X 0,Y 309.101,Z 329.986,A -85,B 0,C 180,E1 14189.263,E2 14189.263} C_VEL
LIN {X 0,Y 311.029,Z 333.796,A -85,B 0,C 180,E1 14187.53,E2 14187.53} C_VEL
LIN {X 0,Y 312.131,Z 336.079,A -85,B 0,C 180,E1 14186.566,E2 14186.566} C_VEL
LIN {X 0,Y 314.327,Z 340.202,A -85,B 0,C 180,E1 14184.847,E2 14184.847} C_VEL
LIN {X 0,Y 316.781,Z 345.256,A -85,B 0,C 180,E1 14182.925,E2 14182.925} C_VEL
LIN {X 0,Y 320.44,Z 352.498,A -85,B 0,C 180,E1 14180.495,E2 14180.495} C_VEL
LIN {X 0,Y 331.091,Z 367.219,A -85,B 0,C 180,E1 14177.55,E2 14177.55} C_VEL
LIN {X 0,Y 340.99,Z 382.18,A -85,B 0,C 180,E1 14175.095,E2 14175.095} C_VEL
LIN {X 0,Y 351.296,Z 399.682,A -85,B 0,C 180,E1 14172.75,E2 14172.75} C_VEL
LIN {X 0,Y 353.779,Z 404.616,A -85,B 0,C 180,E1 14172.201,E2 14172.201} C_VEL
LIN {X 0,Y 347.238,Z 568.111,A -85,B 0,C 180,E1 14168.956,E2 14168.956} C_VEL
LIN {X 0,Y 346.071,Z 587.129,A -85,B 0,C 180,E1 14168.315,E2 14168.315} C_VEL
LIN {X 0,Y 344.189,Z 605.233,A -85,B 0,C 180,E1 14167.434,E2 14167.434} C_VEL
LIN {X 0,Y 341.573,Z 623.392,A -85,B 0,C 180,E1 14166.248,E2 14166.248} C_VEL
LIN {X 0,Y 338.33,Z 640.905,A -85,B 0,C 180,E1 14164.775,E2 14164.775} C_VEL
LIN {X 0,Y 334.605,Z 657.521,A -85,B 0,C 180,E1 14163.016,E2 14163.016} C_VEL
LIN {X 0,Y 330.694,Z 672.638,A -85,B 0,C 180,E1 14161.031,E2 14161.031} C_VEL
LIN {X 0,Y 326.556,Z 686.891,A -85,B 0,C 180,E1 14158.731,E2 14158.731} C_VEL
LIN {X 0,Y 322.412,Z 699.992,A -85,B 0,C 180,E1 14156.127,E2 14156.127} C_VEL
LIN {X 0,Y 318.524,Z 711.511,A -85,B 0,C 180,E1 14153.298,E2 14153.298} C_VEL
LIN {X 0,Y 315.056,Z 721.512,A -85,B 0,C 180,E1 14150.237,E2 14150.237} C_VEL
LIN {X 0,Y 312.075,Z 730.004,A -85,B 0,C 180,E1 14146.951,E2 14146.951} C_VEL
LIN {X 0,Y 309.705,Z 736.955,A -85,B 0,C 180,E1 14143.441,E2 14143.441} C_VEL
LIN {X 0,Y 308.066,Z 742.07,A -85,B 0,C 180,E1 14139.905,E2 14139.905} C_VEL
LIN {X 0,Y 306.982,Z 745.668,A -85,B 0,C 180,E1 14136.17,E2 14136.17} C_VEL
LIN {X 0,Y 306.47,Z 747.558,A -85,B 0,C 180,E1 14132.431,E2 14132.431} C_VEL
LIN {X 0,Y 306.399,Z 747.825,A -85,B 0,C 180,E1 14128.691,E2 14128.691} C_VEL
LIN {X 0,Y 306.762,Z 746.478,A -85,B 0,C 180,E1 14124.951,E2 14124.951} C_VEL
LIN {X 0,Y 307.649,Z 743.458,A -85,B 0,C 180,E1 14121.214,E2 14121.214} C_VEL
LIN {X 0,Y 309.073,Z 738.927,A -85,B 0,C 180,E1 14117.672,E2 14117.672} C_VEL
LIN {X 0,Y 311.188,Z 732.639,A -85,B 0,C 180,E1 14114.151,E2 14114.151} C_VEL
LIN {X 0,Y 313.922,Z 724.857,A -85,B 0,C 180,E1 14110.85,E2 14110.85} C_VEL
LIN {X 0,Y 317.14,Z 715.637,A -85,B 0,C 180,E1 14107.771,E2 14107.771} C_VEL
LIN {X 0,Y 320.789,Z 705.003,A -85,B 0,C 180,E1 14104.92,E2 14104.92} C_VEL
LIN {X 0,Y 324.736,Z 692.945,A -85,B 0,C 180,E1 14102.295,E2 14102.295} C_VEL
LIN {X 0,Y 328.847,Z 679.386,A -85,B 0,C 180,E1 14099.89,E2 14099.89} C_VEL
LIN {X 0,Y 333.022,Z 664.15,A -85,B 0,C 180,E1 14097.696,E2 14097.696} C_VEL
LIN {X 0,Y 334.817,Z 656.929,A -85,B 0,C 180,E1 14096.806,E2 14096.806} C_VEL
LIN {X 0,Y 335.517,Z 650.79,A -85,B 0,C 180,E1 14096.004,E2 14096.004} C_VEL
LIN {X 0,Y 334.288,Z 635.309,A -85,B 0,C 180,E1 14093.815,E2 14093.815} C_VEL
LIN {X 0,Y 334.729,Z 628.688,A -85,B 0,C 180,E1 14093.133,E2 14093.133} C_VEL
LIN {X 0,Y 337.61,Z 610.753,A -85,B 0,C 180,E1 14091.868,E2 14091.868} C_VEL
LIN {X 0,Y 339.875,Z 591.442,A -85,B 0,C 180,E1 14090.848,E2 14090.848} C_VEL
LIN {X 0,Y 341.288,Z 571.739,A -85,B 0,C 180,E1 14090.129,E2 14090.129} C_VEL
LIN {X 0,Y 343.314,Z 519.336,A -85,B 0,C 180,E1 14089.022,E2 14089.022} C_VEL
LIN {X 0,Y 348.016,Z 407.257,A -85,B 0,C 180,E1 14086.776,E2 14086.776} C_VEL
LIN {X 0,Y 338.565,Z 390.76,A -85,B 0,C 180,E1 14084.569,E2 14084.569} C_VEL
LIN {X 0,Y 329.597,Z 376.698,A -85,B 0,C 180,E1 14082.305,E2 14082.305} C_VEL
LIN {X 0,Y 320.047,Z 362.941,A -85,B 0,C 180,E1 14079.651,E2 14079.651} C_VEL
LIN {X 0,Y 312.328,Z 352.662,A -85,B 0,C 180,E1 14077.233,E2 14077.233} C_VEL
LIN {X 0,Y 309.703,Z 347.533,A -85,B 0,C 180,E1 14075.303,E2 14075.303} C_VEL
LIN {X 0,Y 308.074,Z 344.131,A -85,B 0,C 180,E1 14073.934,E2 14073.934} C_VEL
LIN {X 0,Y 305.835,Z 339.709,A -85,B 0,C 180,E1 14071.98,E2 14071.98} C_VEL
LIN {X 0,Y 303.526,Z 335.171,A -85,B 0,C 180,E1 14069.83,E2 14069.83} C_VEL
LIN {X 0,Y 301.465,Z 331.561,A -85,B 0,C 180,E1 14067.882,E2 14067.882} C_VEL
LIN {X 0,Y 300.708,Z 330.163,A -85,B 0,C 180,E1 14067.099,E2 14067.099} C_VEL
LIN {X 0,Y 298.483,Z 326.463,A -85,B 0,C 180,E1 14064.755,E2 14064.755} C_VEL
LIN {X 0,Y 298.286,Z 325.376,A -85,B 0,C 180,E1 14063.929,E2 14063.929} C_VEL
LIN {X 0,Y 298.261,Z 325.297,A -85,B 0,C 180,E1 14059.383,E2 14059.383} C_VEL
LIN {X 0,Y 298.242,Z 325.299,A -85,B 0,C 180,E1 14054.96,E2 14054.96} C_VEL
LIN {X 0,Y 298.241,Z 325.31,A -85,B 0,C 180,E1 14050.235,E2 14050.235} C_VEL
LIN {X 0,Y 298.257,Z 325.335,A -85,B 0,C 180,E1 14045.772,E2 14045.772} C_VEL
LIN {X 0,Y 298.241,Z 325.312,A -85,B 0,C 180,E1 14041.153,E2 14041.153} C_VEL
LIN {X 0,Y 298.226,Z 325.298,A -85,B 0,C 180,E1 14036.733,E2 14036.733} C_VEL
LIN {X 0,Y 298.233,Z 325.299,A -85,B 0,C 180,E1 14032.1,E2 14032.1} C_VEL
LIN {X 0,Y 298.258,Z 325.306,A -85,B 0,C 180,E1 14027.611,E2 14027.611} C_VEL
LIN {X 0,Y 298.273,Z 325.536,A -85,B 0,C 180,E1 14024.644,E2 14024.644} C_VEL
LIN {X 0,Y 300.103,Z 329.523,A -85,B 0,C 180,E1 14022.334,E2 14022.334} C_VEL
LIN {X 0,Y 301.545,Z 331.035,A -85,B 0,C 180,E1 14021.239,E2 14021.239} C_VEL
LIN {X 0,Y 303.231,Z 334.687,A -85,B 0,C 180,E1 14019.542,E2 14019.542} C_VEL
LIN {X 0,Y 304.739,Z 336.709,A -85,B 0,C 180,E1 14018.44,E2 14018.44} C_VEL
LIN {X 0,Y 307.091,Z 340.86,A -85,B 0,C 180,E1 14016.596,E2 14016.596} C_VEL
LIN {X 0,Y 310.57,Z 347.397,A -85,B 0,C 180,E1 14014.034,E2 14014.034} C_VEL
LIN {X 0,Y 313.239,Z 352.438,A -85,B 0,C 180,E1 14012.223,E2 14012.223} C_VEL
LIN {X 0,Y 317.212,Z 359.983,A -85,B 0,C 180,E1 14009.714,E2 14009.714} C_VEL
LIN {X 0,Y 322.945,Z 371.883,A -85,B 0,C 180,E1 14006.345,E2 14006.345} C_VEL
LIN {X 0,Y 324.709,Z 375.399,A -85,B 0,C 180,E1 14005.542,E2 14005.542} C_VEL
LIN {X 0,Y 334.641,Z 391.162,A -85,B 0,C 180,E1 14002.876,E2 14002.876} C_VEL
LIN {X 0,Y 343.495,Z 406.642,A -85,B 0,C 180,E1 14000.694,E2 14000.694} C_VEL
LIN {X 0,Y 347.369,Z 414.352,A -85,B 0,C 180,E1 13999.772,E2 13999.772} C_VEL
LIN {X 0,Y 348.517,Z 435.646,A -85,B 0,C 180,E1 13998.919,E2 13998.919} C_VEL
LIN {X 0,Y 338.522,Z 627.448,A -85,B 0,C 180,E1 13994.676,E2 13994.676} C_VEL
LIN {X 0,Y 336.163,Z 649.336,A -85,B 0,C 180,E1 13993.925,E2 13993.925} C_VEL
LIN {X 0,Y 332.862,Z 670.114,A -85,B 0,C 180,E1 13992.929,E2 13992.929} C_VEL
LIN {X 0,Y 328.796,Z 690.948,A -85,B 0,C 180,E1 13991.576,E2 13991.576} C_VEL
LIN {X 0,Y 324.522,Z 710.006,A -85,B 0,C 180,E1 13989.969,E2 13989.969} C_VEL
LIN {X 0,Y 319.911,Z 728.609,A -85,B 0,C 180,E1 13988.002,E2 13988.002} C_VEL
LIN {X 0,Y 315.591,Z 744.93,A -85,B 0,C 180,E1 13985.881,E2 13985.881} C_VEL
LIN {X 0,Y 311.177,Z 761.167,A -85,B 0,C 180,E1 13983.328,E2 13983.328} C_VEL
LIN {X 0,Y 307.169,Z 775.974,A -85,B 0,C 180,E1 13980.516,E2 13980.516} C_VEL
LIN {X 0,Y 303.504,Z 790.188,A -85,B 0,C 180,E1 13977.252,E2 13977.252} C_VEL
LIN {X 0,Y 300.59,Z 802.793,A -85,B 0,C 180,E1 13973.733,E2 13973.733} C_VEL
LIN {X 0,Y 298.623,Z 813.259,A -85,B 0,C 180,E1 13970.173,E2 13970.173} C_VEL
LIN {X 0,Y 297.44,Z 822.245,A -85,B 0,C 180,E1 13966.401,E2 13966.401} C_VEL
LIN {X 0,Y 296.992,Z 829.303,A -85,B 0,C 180,E1 13962.64,E2 13962.64} C_VEL
LIN {X 0,Y 297.099,Z 834.231,A -85,B 0,C 180,E1 13959.101,E2 13959.101} C_VEL
LIN {X 0,Y 297.429,Z 837.601,A -85,B 0,C 180,E1 13955.594,E2 13955.594} C_VEL
LIN {X 0,Y 297.723,Z 839.363,A -85,B 0,C 180,E1 13952.31,E2 13952.31} C_VEL
LIN {X 0,Y 297.792,Z 839.616,A -85,B 0,C 180,E1 13949.038,E2 13949.038} C_VEL
LIN {X 0,Y 297.566,Z 838.527,A -85,B 0,C 180,E1 13945.761,E2 13945.761} C_VEL
LIN {X 0,Y 297.233,Z 835.907,A -85,B 0,C 180,E1 13942.462,E2 13942.462} C_VEL
LIN {X 0,Y 296.994,Z 831.363,A -85,B 0,C 180,E1 13938.74,E2 13938.74} C_VEL
LIN {X 0,Y 297.205,Z 825.031,A -85,B 0,C 180,E1 13934.987,E2 13934.987} C_VEL
LIN {X 0,Y 298.078,Z 816.808,A -85,B 0,C 180,E1 13931.216,E2 13931.216} C_VEL
LIN {X 0,Y 299.838,Z 806.52,A -85,B 0,C 180,E1 13927.451,E2 13927.451} C_VEL
LIN {X 0,Y 302.426,Z 794.641,A -85,B 0,C 180,E1 13923.915,E2 13923.915} C_VEL
LIN {X 0,Y 305.758,Z 781.237,A -85,B 0,C 180,E1 13920.627,E2 13920.627} C_VEL
LIN {X 0,Y 309.764,Z 766.307,A -85,B 0,C 180,E1 13917.602,E2 13917.602} C_VEL
LIN {X 0,Y 313.918,Z 750.922,A -85,B 0,C 180,E1 13915.019,E2 13915.019} C_VEL
LIN {X 0,Y 318.404,Z 734.168,A -85,B 0,C 180,E1 13912.696,E2 13912.696} C_VEL
LIN {X 0,Y 323.05,Z 715.791,A -85,B 0,C 180,E1 13910.619,E2 13910.619} C_VEL
LIN {X 0,Y 327.542,Z 696.359,A -85,B 0,C 180,E1 13908.866,E2 13908.866} C_VEL
LIN {X 0,Y 331.503,Z 677.008,A -85,B 0,C 180,E1 13907.5,E2 13907.5} C_VEL
LIN {X 0,Y 334.931,Z 657.164,A -85,B 0,C 180,E1 13906.433,E2 13906.433} C_VEL
LIN {X 0,Y 337.6,Z 636.588,A -85,B 0,C 180,E1 13905.621,E2 13905.621} C_VEL
LIN {X 0,Y 339.243,Z 614.759,A -85,B 0,C 180,E1 13905.024,E2 13905.024} C_VEL
LIN {X 0,Y 348.464,Z 433.38,A -85,B 0,C 180,E1 13901.034,E2 13901.034} C_VEL
LIN {X 0,Y 347.056,Z 413.552,A -85,B 0,C 180,E1 13900.191,E2 13900.191} C_VEL
LIN {X 0,Y 338.3,Z 397.503,A -85,B 0,C 180,E1 13898.095,E2 13898.095} C_VEL
LIN {X 0,Y 328.678,Z 381.539,A -85,B 0,C 180,E1 13895.603,E2 13895.603} C_VEL
LIN {X 0,Y 323.71,Z 373.599,A -85,B 0,C 180,E1 13894.131,E2 13894.131} C_VEL
LIN {X 0,Y 318.309,Z 362.299,A -85,B 0,C 180,E1 13891.007,E2 13891.007} C_VEL
LIN {X 0,Y 313.987,Z 353.863,A -85,B 0,C 180,E1 13888.325,E2 13888.325} C_VEL
LIN {X 0,Y 311.504,Z 349.228,A -85,B 0,C 180,E1 13886.703,E2 13886.703} C_VEL
LIN {X 0,Y 309.417,Z 345.303,A -85,B 0,C 180,E1 13885.248,E2 13885.248} C_VEL
LIN {X 0,Y 306.965,Z 340.727,A -85,B 0,C 180,E1 13883.414,E2 13883.414} C_VEL
LIN {X 0,Y 304.831,Z 336.987,A -85,B 0,C 180,E1 13881.755,E2 13881.755} C_VEL
LIN {X 0,Y 303.891,Z 335.482,A -85,B 0,C 180,E1 13881.016,E2 13881.016} C_VEL
LIN {X 0,Y 301.737,Z 331.756,A -85,B 0,C 180,E1 13879.15,E2 13879.15} C_VEL
LIN {X 0,Y 300.935,Z 330.339,A -85,B 0,C 180,E1 13878.399,E2 13878.399} C_VEL
LIN {X 0,Y 298.671,Z 327.035,A -85,B 0,C 180,E1 13876.332,E2 13876.332} C_VEL
LIN {X 0,Y 298.264,Z 325.446,A -85,B 0,C 180,E1 13875.356,E2 13875.356} C_VEL
LIN {X 0,Y 298.261,Z 325.333,A -85,B 0,C 180,E1 13870.82,E2 13870.82} C_VEL
LIN {X 0,Y 298.26,Z 325.316,A -85,B 0,C 180,E1 13866.351,E2 13866.351} C_VEL
LIN {X 0,Y 298.227,Z 325.305,A -85,B 0,C 180,E1 13861.729,E2 13861.729} C_VEL
LIN {X 0,Y 298.225,Z 325.298,A -85,B 0,C 180,E1 13857.117,E2 13857.117} C_VEL
LIN {X 0,Y 298.248,Z 325.305,A -85,B 0,C 180,E1 13852.681,E2 13852.681} C_VEL
LIN {X 0,Y 298.258,Z 325.33,A -85,B 0,C 180,E1 13848.196,E2 13848.196} C_VEL
LIN {X 0,Y 298.244,Z 325.321,A -85,B 0,C 180,E1 13843.643,E2 13843.643} C_VEL
LIN {X 0,Y 298.245,Z 325.309,A -85,B 0,C 180,E1 13838.978,E2 13838.978} C_VEL
LIN {X 0,Y 298.291,Z 325.596,A -85,B 0,C 180,E1 13835.545,E2 13835.545} C_VEL
LIN {X 0,Y 300.232,Z 329.679,A -85,B 0,C 180,E1 13833.068,E2 13833.068} C_VEL
LIN {X 0,Y 301.324,Z 331.131,A -85,B 0,C 180,E1 13832.104,E2 13832.104} C_VEL
LIN {X 0,Y 303.026,Z 334.6,A -85,B 0,C 180,E1 13830.334,E2 13830.334} C_VEL
LIN {X 0,Y 304.139,Z 336.451,A -85,B 0,C 180,E1 13829.365,E2 13829.365} C_VEL
LIN {X 0,Y 306.759,Z 341.521,A -85,B 0,C 180,E1 13827.021,E2 13827.021} C_VEL
LIN {X 0,Y 309.09,Z 346.172,A -85,B 0,C 180,E1 13825.07,E2 13825.07} C_VEL
LIN {X 0,Y 312.683,Z 353.174,A -85,B 0,C 180,E1 13822.467,E2 13822.467} C_VEL
LIN {X 0,Y 321.163,Z 364.628,A -85,B 0,C 180,E1 13819.876,E2 13819.876} C_VEL
LIN {X 0,Y 330.578,Z 378.201,A -85,B 0,C 180,E1 13817.303,E2 13817.303} C_VEL
LIN {X 0,Y 340.215,Z 393.56,A -85,B 0,C 180,E1 13814.905,E2 13814.905} C_VEL
LIN {X 0,Y 348.072,Z 407.676,A -85,B 0,C 180,E1 13813.08,E2 13813.08} C_VEL
LIN {X 0,Y 341.306,Z 568.746,A -85,B 0,C 180,E1 13809.843,E2 13809.843} C_VEL
LIN {X 0,Y 340.081,Z 587.888,A -85,B 0,C 180,E1 13809.191,E2 13809.191} C_VEL
LIN {X 0,Y 338.085,Z 606.306,A -85,B 0,C 180,E1 13808.284,E2 13808.284} C_VEL
LIN {X 0,Y 335.455,Z 623.878,A -85,B 0,C 180,E1 13807.125,E2 13807.125} C_VEL
LIN {X 0,Y 332.137,Z 641.248,A -85,B 0,C 180,E1 13805.656,E2 13805.656} C_VEL
LIN {X 0,Y 328.255,Z 657.979,A -85,B 0,C 180,E1 13803.876,E2 13803.876} C_VEL
LIN {X 0,Y 324.125,Z 673.382,A -85,B 0,C 180,E1 13801.836,E2 13801.836} C_VEL
LIN {X 0,Y 319.951,Z 687.213,A -85,B 0,C 180,E1 13799.587,E2 13799.587} C_VEL
LIN {X 0,Y 315.6,Z 700.452,A -85,B 0,C 180,E1 13796.938,E2 13796.938} C_VEL
LIN {X 0,Y 311.501,Z 712.095,A -85,B 0,C 180,E1 13794.056,E2 13794.056} C_VEL
LIN {X 0,Y 307.822,Z 722.207,A -85,B 0,C 180,E1 13790.934,E2 13790.934} C_VEL
LIN {X 0,Y 304.651,Z 730.8,A -85,B 0,C 180,E1 13787.574,E2 13787.574} C_VEL
LIN {X 0,Y 302.105,Z 737.845,A -85,B 0,C 180,E1 13783.981,E2 13783.981} C_VEL
LIN {X 0,Y 300.335,Z 743.048,A -85,B 0,C 180,E1 13780.356,E2 13780.356} C_VEL
LIN {X 0,Y 299.151,Z 746.729,A -85,B 0,C 180,E1 13776.525,E2 13776.525} C_VEL
LIN {X 0,Y 298.579,Z 748.7,A -85,B 0,C 180,E1 13772.687,E2 13772.687} C_VEL
LIN {X 0,Y 298.487,Z 749.045,A -85,B 0,C 180,E1 13768.848,E2 13768.848} C_VEL
LIN {X 0,Y 298.845,Z 747.781,A -85,B 0,C 180,E1 13765.01,E2 13765.01} C_VEL
LIN {X 0,Y 299.756,Z 744.849,A -85,B 0,C 180,E1 13761.174,E2 13761.174} C_VEL
LIN {X 0,Y 301.233,Z 740.412,A -85,B 0,C 180,E1 13757.541,E2 13757.541} C_VEL
LIN {X 0,Y 303.425,Z 734.224,A -85,B 0,C 180,E1 13753.931,E2 13753.931} C_VEL
LIN {X 0,Y 306.26,Z 726.554,A -85,B 0,C 180,E1 13750.549,E2 13750.549} C_VEL
LIN {X 0,Y 309.598,Z 717.462,A -85,B 0,C 180,E1 13747.399,E2 13747.399} C_VEL
LIN {X 0,Y 313.635,Z 706.249,A -85,B 0,C 180,E1 13744.307,E2 13744.307} C_VEL
LIN {X 0,Y 317.755,Z 694.212,A -85,B 0,C 180,E1 13741.632,E2 13741.632} C_VEL
LIN {X 0,Y 322.118,Z 680.418,A -85,B 0,C 180,E1 13739.141,E2 13739.141} C_VEL
LIN {X 0,Y 326.383,Z 665.492,A -85,B 0,C 180,E1 13736.956,E2 13736.956} C_VEL
LIN {X 0,Y 330.298,Z 649.867,A -85,B 0,C 180,E1 13735.102,E2 13735.102} C_VEL
LIN {X 0,Y 334.018,Z 632.337,A -85,B 0,C 180,E1 13733.439,E2 13733.439} C_VEL
LIN {X 0,Y 334.729,Z 628.688,A -85,B 0,C 180,E1 13733.133,E2 13733.133} C_VEL
LIN {X 0,Y 335.223,Z 621.912,A -85,B 0,C 180,E1 13732.488,E2 13732.488} C_VEL
LIN {X 0,Y 333.336,Z 605.824,A -85,B 0,C 180,E1 13730.785,E2 13730.785} C_VEL
LIN {X 0,Y 333.268,Z 598.698,A -85,B 0,C 180,E1 13730.261,E2 13730.261} C_VEL
LIN {X 0,Y 333.358,Z 597.642,A -85,B 0,C 180,E1 13730.205,E2 13730.205} C_VEL
LIN {X 0,Y 335.063,Z 578.214,A -85,B 0,C 180,E1 13729.399,E2 13729.399} C_VEL
LIN {X 0,Y 336.115,Z 554.132,A -85,B 0,C 180,E1 13728.778,E2 13728.778} C_VEL
LIN {X 0,Y 342.447,Z 410.601,A -85,B 0,C 180,E1 13725.881,E2 13725.881} C_VEL
LIN {X 0,Y 332.833,Z 393.769,A -85,B 0,C 180,E1 13723.527,E2 13723.527} C_VEL
LIN {X 0,Y 323.264,Z 378.915,A -85,B 0,C 180,E1 13720.975,E2 13720.975} C_VEL
LIN {X 0,Y 313.207,Z 364.634,A -85,B 0,C 180,E1 13717.976,E2 13717.976} C_VEL
LIN {X 0,Y 304.622,Z 353.575,A -85,B 0,C 180,E1 13715.058,E2 13715.058} C_VEL
LIN {X 0,Y 302.664,Z 349.691,A -85,B 0,C 180,E1 13713.483,E2 13713.483} C_VEL
LIN {X 0,Y 300.659,Z 345.658,A -85,B 0,C 180,E1 13711.698,E2 13711.698} C_VEL
LIN {X 0,Y 298.421,Z 341.198,A -85,B 0,C 180,E1 13709.507,E2 13709.507} C_VEL
LIN {X 0,Y 296.48,Z 337.511,A -85,B 0,C 180,E1 13707.511,E2 13707.511} C_VEL
LIN {X 0,Y 293.618,Z 332.441,A -85,B 0,C 180,E1 13704.334,E2 13704.334} C_VEL
LIN {X 0,Y 292.341,Z 330.711,A -85,B 0,C 180,E1 13702.949,E2 13702.949} C_VEL
LIN {X 0,Y 290.377,Z 326.58,A -85,B 0,C 180,E1 13699.722,E2 13699.722} C_VEL
LIN {X 0,Y 290.32,Z 326.289,A -85,B 0,C 180,E1 13695.358,E2 13695.358} C_VEL
LIN {X 0,Y 290.297,Z 326.308,A -85,B 0,C 180,E1 13690.719,E2 13690.719} C_VEL
LIN {X 0,Y 290.301,Z 326.318,A -85,B 0,C 180,E1 13686.13,E2 13686.13} C_VEL
LIN {X 0,Y 290.313,Z 326.291,A -85,B 0,C 180,E1 13681.579,E2 13681.579} C_VEL
LIN {X 0,Y 290.297,Z 326.283,A -85,B 0,C 180,E1 13677.039,E2 13677.039} C_VEL
LIN {X 0,Y 290.29,Z 326.29,A -85,B 0,C 180,E1 13672.48,E2 13672.48} C_VEL
LIN {X 0,Y 290.362,Z 326.628,A -85,B 0,C 180,E1 13669.083,E2 13669.083} C_VEL
LIN {X 0,Y 292.426,Z 330.794,A -85,B 0,C 180,E1 13665.951,E2 13665.951} C_VEL
LIN {X 0,Y 293.803,Z 332.415,A -85,B 0,C 180,E1 13664.607,E2 13664.607} C_VEL
LIN {X 0,Y 295.909,Z 336.401,A -85,B 0,C 180,E1 13662.296,E2 13662.296} C_VEL
LIN {X 0,Y 296.9,Z 337.395,A -85,B 0,C 180,E1 13661.545,E2 13661.545} C_VEL
LIN {X 0,Y 298.811,Z 341.358,A -85,B 0,C 180,E1 13659.636,E2 13659.636} C_VEL
LIN {X 0,Y 300.03,Z 343.088,A -85,B 0,C 180,E1 13658.701,E2 13658.701} C_VEL
LIN {X 0,Y 303.003,Z 348.659,A -85,B 0,C 180,E1 13656.261,E2 13656.261} C_VEL
LIN {X 0,Y 305.756,Z 353.796,A -85,B 0,C 180,E1 13654.22,E2 13654.22} C_VEL
LIN {X 0,Y 309.863,Z 361.613,A -85,B 0,C 180,E1 13651.361,E2 13651.361} C_VEL
LIN {X 0,Y 315.892,Z 373.809,A -85,B 0,C 180,E1 13647.716,E2 13647.716} C_VEL
LIN {X 0,Y 324.972,Z 387.721,A -85,B 0,C 180,E1 13645.038,E2 13645.038} C_VEL
LIN {X 0,Y 334.512,Z 403.802,A -85,B 0,C 180,E1 13642.482,E2 13642.482} C_VEL
LIN {X 0,Y 341.977,Z 417.8,A -85,B 0,C 180,E1 13640.621,E2 13640.621} C_VEL
LIN {X 0,Y 342.894,Z 436.769,A -85,B 0,C 180,E1 13639.851,E2 13639.851} C_VEL
LIN {X 0,Y 332.625,Z 626.475,A -85,B 0,C 180,E1 13635.614,E2 13635.614} C_VEL
LIN {X 0,Y 330.213,Z 648.278,A -85,B 0,C 180,E1 13634.861,E2 13634.861} C_VEL
LIN {X 0,Y 326.821,Z 669.02,A -85,B 0,C 180,E1 13633.862,E2 13633.862} C_VEL
LIN {X 0,Y 322.839,Z 688.695,A -85,B 0,C 180,E1 13632.586,E2 13632.586} C_VEL
LIN {X 0,Y 318.472,Z 707.543,A -85,B 0,C 180,E1 13631.007,E2 13631.007} C_VEL
LIN {X 0,Y 313.842,Z 725.625,A -85,B 0,C 180,E1 13629.108,E2 13629.108} C_VEL
LIN {X 0,Y 309.037,Z 743.042,A -85,B 0,C 180,E1 13626.852,E2 13626.852} C_VEL
LIN {X 0,Y 304.41,Z 759.264,A -85,B 0,C 180,E1 13624.284,E2 13624.284} C_VEL
LIN {X 0,Y 300.01,Z 774.636,A -85,B 0,C 180,E1 13621.325,E2 13621.325} C_VEL
LIN {X 0,Y 296.308,Z 788.111,A -85,B 0,C 180,E1 13618.19,E2 13618.19} C_VEL
LIN {X 0,Y 293.28,Z 800.234,A -85,B 0,C 180,E1 13614.792,E2 13614.792} C_VEL
LIN {X 0,Y 291.041,Z 810.954,A -85,B 0,C 180,E1 13611.144,E2 13611.144} C_VEL
LIN {X 0,Y 289.627,Z 820.148,A -85,B 0,C 180,E1 13607.27,E2 13607.27} C_VEL
LIN {X 0,Y 289.057,Z 827.365,A -85,B 0,C 180,E1 13603.4,E2 13603.4} C_VEL
LIN {X 0,Y 289.113,Z 832.759,A -85,B 0,C 180,E1 13599.555,E2 13599.555} C_VEL
LIN {X 0,Y 289.472,Z 836.309,A -85,B 0,C 180,E1 13595.863,E2 13595.863} C_VEL
LIN {X 0,Y 289.794,Z 838.08,A -85,B 0,C 180,E1 13592.571,E2 13592.571} C_VEL
LIN {X 0,Y 289.886,Z 838.441,A -85,B 0,C 180,E1 13589.209,E2 13589.209} C_VEL
LIN {X 0,Y 289.668,Z 837.477,A -85,B 0,C 180,E1 13585.987,E2 13585.987} C_VEL
LIN {X 0,Y 289.291,Z 834.873,A -85,B 0,C 180,E1 13582.453,E2 13582.453} C_VEL
LIN {X 0,Y 289.03,Z 830.708,A -85,B 0,C 180,E1 13578.83,E2 13578.83} C_VEL
LIN {X 0,Y 289.219,Z 824.56,A -85,B 0,C 180,E1 13574.973,E2 13574.973} C_VEL
LIN {X 0,Y 290.106,Z 816.47,A -85,B 0,C 180,E1 13571.097,E2 13571.097} C_VEL
LIN {X 0,Y 291.797,Z 806.944,A -85,B 0,C 180,E1 13567.433,E2 13567.433} C_VEL
LIN {X 0,Y 294.417,Z 795.415,A -85,B 0,C 180,E1 13563.802,E2 13563.802} C_VEL
LIN {X 0,Y 297.853,Z 782.251,A -85,B 0,C 180,E1 13560.392,E2 13560.392} C_VEL
LIN {X 0,Y 302.056,Z 767.37,A -85,B 0,C 180,E1 13557.222,E2 13557.222} C_VEL
LIN {X 0,Y 306.64,Z 751.293,A -85,B 0,C 180,E1 13554.408,E2 13554.408} C_VEL
LIN {X 0,Y 311.475,Z 734.13,A -85,B 0,C 180,E1 13551.952,E2 13551.952} C_VEL
LIN {X 0,Y 316.088,Z 716.815,A -85,B 0,C 180,E1 13549.932,E2 13549.932} C_VEL
LIN {X 0,Y 320.628,Z 698.246,A -85,B 0,C 180,E1 13548.185,E2 13548.185} C_VEL
LIN {X 0,Y 324.793,Z 679.161,A -85,B 0,C 180,E1 13546.769,E2 13546.769} C_VEL
LIN {X 0,Y 328.496,Z 659.002,A -85,B 0,C 180,E1 13545.631,E2 13545.631} C_VEL
LIN {X 0,Y 331.501,Z 637.353,A -85,B 0,C 180,E1 13544.742,E2 13544.742} C_VEL
LIN {X 0,Y 333.284,Z 615.358,A -85,B 0,C 180,E1 13544.119,E2 13544.119} C_VEL
LIN {X 0,Y 342.847,Z 434.463,A -85,B 0,C 180,E1 13540.101,E2 13540.101} C_VEL
LIN {X 0,Y 341.646,Z 417.212,A -85,B 0,C 180,E1 13539.343,E2 13539.343} C_VEL
LIN {X 0,Y 332.368,Z 400.123,A -85,B 0,C 180,E1 13537.015,E2 13537.015} C_VEL
LIN {X 0,Y 323.108,Z 384.877,A -85,B 0,C 180,E1 13534.492,E2 13534.492} C_VEL
LIN {X 0,Y 315.51,Z 373.117,A -85,B 0,C 180,E1 13532.167,E2 13532.167} C_VEL
LIN {X 0,Y 309.723,Z 361.189,A -85,B 0,C 180,E1 13528.54,E2 13528.54} C_VEL
LIN {X 0,Y 304.664,Z 351.646,A -85,B 0,C 180,E1 13525.046,E2 13525.046} C_VEL
LIN {X 0,Y 301.904,Z 346.675,A -85,B 0,C 180,E1 13522.976,E2 13522.976} C_VEL
LIN {X 0,Y 299.449,Z 342.125,A -85,B 0,C 180,E1 13520.932,E2 13520.932} C_VEL
LIN {X 0,Y 297.074,Z 338.101,A -85,B 0,C 180,E1 13518.85,E2 13518.85} C_VEL
LIN {X 0,Y 296.51,Z 336.975,A -85,B 0,C 180,E1 13518.276,E2 13518.276} C_VEL
LIN {X 0,Y 294.245,Z 333.717,A -85,B 0,C 180,E1 13516.179,E2 13516.179} C_VEL
LIN {X 0,Y 293.336,Z 331.648,A -85,B 0,C 180,E1 13515.013,E2 13515.013} C_VEL
LIN {X 0,Y 290.735,Z 328.06,A -85,B 0,C 180,E1 13512.109,E2 13512.109} C_VEL
LIN {X 0,Y 290.339,Z 326.466,A -85,B 0,C 180,E1 13510.918,E2 13510.918} C_VEL
LIN {X 0,Y 290.33,Z 326.299,A -85,B 0,C 180,E1 13506.525,E2 13506.525} C_VEL
LIN {X 0,Y 290.295,Z 326.289,A -85,B 0,C 180,E1 13501.973,E2 13501.973} C_VEL
LIN {X 0,Y 290.281,Z 326.288,A -85,B 0,C 180,E1 13497.433,E2 13497.433} C_VEL
LIN {X 0,Y 290.299,Z 326.298,A -85,B 0,C 180,E1 13492.877,E2 13492.877} C_VEL
LIN {X 0,Y 290.32,Z 326.319,A -85,B 0,C 180,E1 13488.276,E2 13488.276} C_VEL
LIN {X 0,Y 290.31,Z 326.304,A -85,B 0,C 180,E1 13483.801,E2 13483.801} C_VEL
LIN {X 0,Y 290.365,Z 326.591,A -85,B 0,C 180,E1 13479.973,E2 13479.973} C_VEL
LIN {X 0,Y 292.309,Z 330.67,A -85,B 0,C 180,E1 13476.836,E2 13476.836} C_VEL
LIN {X 0,Y 293.589,Z 332.42,A -85,B 0,C 180,E1 13475.449,E2 13475.449} C_VEL
LIN {X 0,Y 295.674,Z 336.283,A -85,B 0,C 180,E1 13473.054,E2 13473.054} C_VEL
LIN {X 0,Y 296.465,Z 337.573,A -85,B 0,C 180,E1 13472.262,E2 13472.262} C_VEL
LIN {X 0,Y 298.639,Z 341.479,A -85,B 0,C 180,E1 13470.126,E2 13470.126} C_VEL
LIN {X 0,Y 301.629,Z 347.502,A -85,B 0,C 180,E1 13467.294,E2 13467.294} C_VEL
LIN {X 0,Y 304.135,Z 352.694,A -85,B 0,C 180,E1 13465.107,E2 13465.107} C_VEL
LIN {X 0,Y 306.245,Z 355.597,A -85,B 0,C 180,E1 13464.18,E2 13464.18} C_VEL
LIN {X 0,Y 314.388,Z 366.42,A -85,B 0,C 180,E1 13461.497,E2 13461.497} C_VEL
LIN {X 0,Y 323.76,Z 379.679,A -85,B 0,C 180,E1 13458.749,E2 13458.749} C_VEL
LIN {X 0,Y 333.437,Z 394.86,A -85,B 0,C 180,E1 13456.186,E2 13456.186} C_VEL
LIN {X 0,Y 342.449,Z 410.811,A -85,B 0,C 180,E1 13453.988,E2 13453.988} C_VEL
LIN {X 0,Y 335.457,Z 569.4,A -85,B 0,C 180,E1 13450.76,E2 13450.76} C_VEL
LIN {X 0,Y 334.185,Z 588.515,A -85,B 0,C 180,E1 13450.104,E2 13450.104} C_VEL
LIN {X 0,Y 332.059,Z 607.376,A -85,B 0,C 180,E1 13449.165,E2 13449.165} C_VEL
LIN {X 0,Y 329.274,Z 625.188,A -85,B 0,C 180,E1 13447.971,E2 13447.971} C_VEL
LIN {X 0,Y 325.721,Z 642.956,A -85,B 0,C 180,E1 13446.439,E2 13446.439} C_VEL
LIN {X 0,Y 321.742,Z 659.358,A -85,B 0,C 180,E1 13444.658,E2 13444.658} C_VEL
LIN {X 0,Y 317.359,Z 675.002,A -85,B 0,C 180,E1 13442.543,E2 13442.543} C_VEL
LIN {X 0,Y 313.103,Z 688.498,A -85,B 0,C 180,E1 13440.301,E2 13440.301} C_VEL
LIN {X 0,Y 308.567,Z 701.711,A -85,B 0,C 180,E1 13437.604,E2 13437.604} C_VEL
LIN {X 0,Y 304.284,Z 713.336,A -85,B 0,C 180,E1 13434.664,E2 13434.664} C_VEL
LIN {X 0,Y 300.429,Z 723.435,A -85,B 0,C 180,E1 13431.474,E2 13431.474} C_VEL
LIN {X 0,Y 297.099,Z 732.018,A -85,B 0,C 180,E1 13428.036,E2 13428.036} C_VEL
LIN {X 0,Y 294.413,Z 739.058,A -85,B 0,C 180,E1 13424.354,E2 13424.354} C_VEL
LIN {X 0,Y 292.54,Z 744.256,A -85,B 0,C 180,E1 13420.635,E2 13420.635} C_VEL
LIN {X 0,Y 291.285,Z 747.933,A -85,B 0,C 180,E1 13416.702,E2 13416.702} C_VEL
LIN {X 0,Y 290.676,Z 749.902,A -85,B 0,C 180,E1 13412.76,E2 13412.76} C_VEL
LIN {X 0,Y 290.578,Z 750.247,A -85,B 0,C 180,E1 13408.817,E2 13408.817} C_VEL
LIN {X 0,Y 290.961,Z 748.983,A -85,B 0,C 180,E1 13404.874,E2 13404.874} C_VEL
LIN {X 0,Y 291.928,Z 746.053,A -85,B 0,C 180,E1 13400.936,E2 13400.936} C_VEL
LIN {X 0,Y 293.492,Z 741.62,A -85,B 0,C 180,E1 13397.207,E2 13397.207} C_VEL
LIN {X 0,Y 295.809,Z 735.438,A -85,B 0,C 180,E1 13393.506,E2 13393.506} C_VEL
LIN {X 0,Y 298.793,Z 727.774,A -85,B 0,C 180,E1 13390.043,E2 13390.043} C_VEL
LIN {X 0,Y 302.523,Z 718.097,A -85,B 0,C 180,E1 13386.634,E2 13386.634} C_VEL
LIN {X 0,Y 306.519,Z 707.492,A -85,B 0,C 180,E1 13383.665,E2 13383.665} C_VEL
LIN {X 0,Y 310.818,Z 695.477,A -85,B 0,C 180,E1 13380.94,E2 13380.94} C_VEL
LIN {X 0,Y 315.28,Z 681.98,A -85,B 0,C 180,E1 13378.449,E2 13378.449} C_VEL
LIN {X 0,Y 319.801,Z 666.833,A -85,B 0,C 180,E1 13376.186,E2 13376.186} C_VEL
LIN {X 0,Y 324.039,Z 650.566,A -85,B 0,C 180,E1 13374.229,E2 13374.229} C_VEL
LIN {X 0,Y 327.734,Z 633.843,A -85,B 0,C 180,E1 13372.62,E2 13372.62} C_VEL
LIN {X 0,Y 330.992,Z 615.43,A -85,B 0,C 180,E1 13371.228,E2 13371.228} C_VEL
LIN {X 0,Y 333.358,Z 597.642,A -85,B 0,C 180,E1 13370.205,E2 13370.205} C_VEL
LIN {X 0,Y 333.417,Z 590.341,A -85,B 0,C 180,E1 13369.748,E2 13369.748} C_VEL
LIN {X 0,Y 330.472,Z 572.138,A -85,B 0,C 180,E1 13368.365,E2 13368.365} C_VEL
LIN {X 0,Y 330.034,Z 564.642,A -85,B 0,C 180,E1 13368.039,E2 13368.039} C_VEL
LIN {X 0,Y 336.89,Z 413.857,A -85,B 0,C 180,E1 13364.94,E2 13364.94} C_VEL
LIN {X 0,Y 327.682,Z 397.794,A -85,B 0,C 180,E1 13362.581,E2 13362.581} C_VEL
LIN {X 0,Y 318.487,Z 383.339,A -85,B 0,C 180,E1 13360.005,E2 13360.005} C_VEL
LIN {X 0,Y 309.533,Z 370.652,A -85,B 0,C 180,E1 13357.219,E2 13357.219} C_VEL
LIN {X 0,Y 302.01,Z 360.764,A -85,B 0,C 180,E1 13354.596,E2 13354.596} C_VEL
LIN {X 0,Y 296.797,Z 354.105,A -85,B 0,C 180,E1 13352.502,E2 13352.502} C_VEL
LIN {X 0,Y 295.354,Z 351.3,A -85,B 0,C 180,E1 13351.195,E2 13351.195} C_VEL
LIN {X 0,Y 293.337,Z 347.235,A -85,B 0,C 180,E1 13349.172,E2 13349.172} C_VEL
LIN {X 0,Y 291.114,Z 342.876,A -85,B 0,C 180,E1 13346.74,E2 13346.74} C_VEL
LIN {X 0,Y 288.896,Z 338.832,A -85,B 0,C 180,E1 13344.104,E2 13344.104} C_VEL
LIN {X 0,Y 287.834,Z 337.317,A -85,B 0,C 180,E1 13342.896,E2 13342.896} C_VEL
LIN {X 0,Y 285.304,Z 332.559,A -85,B 0,C 180,E1 13339.022,E2 13339.022} C_VEL
LIN {X 0,Y 282.392,Z 327.522,A -85,B 0,C 180,E1 13332.474,E2 13332.474} C_VEL
LIN {X 0,Y 282.37,Z 327.274,A -85,B 0,C 180,E1 13327.938,E2 13327.938} C_VEL
LIN {X 0,Y 282.37,Z 327.272,A -85,B 0,C 180,E1 13323.452,E2 13323.452} C_VEL
LIN {X 0,Y 282.348,Z 327.285,A -85,B 0,C 180,E1 13318.783,E2 13318.783} C_VEL
LIN {X 0,Y 282.425,Z 327.72,A -85,B 0,C 180,E1 13315.94,E2 13315.94} C_VEL
LIN {X 0,Y 285.978,Z 333.412,A -85,B 0,C 180,E1 13309.118,E2 13309.118} C_VEL
LIN {X 0,Y 288.041,Z 337.427,A -85,B 0,C 180,E1 13306.142,E2 13306.142} C_VEL
LIN {X 0,Y 289.259,Z 338.729,A -85,B 0,C 180,E1 13304.975,E2 13304.975} C_VEL
LIN {X 0,Y 291.325,Z 342.844,A -85,B 0,C 180,E1 13302.573,E2 13302.573} C_VEL
LIN {X 0,Y 292.38,Z 344.211,A -85,B 0,C 180,E1 13301.663,E2 13301.663} C_VEL
LIN {X 0,Y 294.621,Z 348.323,A -85,B 0,C 180,E1 13299.54,E2 13299.54} C_VEL
LIN {X 0,Y 298.029,Z 354.529,A -85,B 0,C 180,E1 13296.68,E2 13296.68} C_VEL
LIN {X 0,Y 300.849,Z 360.107,A -85,B 0,C 180,E1 13294.403,E2 13294.403} C_VEL
LIN {X 0,Y 304.889,Z 367.816,A -85,B 0,C 180,E1 13291.608,E2 13291.608} C_VEL
LIN {X 0,Y 307.814,Z 373.49,A -85,B 0,C 180,E1 13289.878,E2 13289.878} C_VEL
LIN {X 0,Y 316.729,Z 386.607,A -85,B 0,C 180,E1 13287.006,E2 13287.006} C_VEL
LIN {X 0,Y 326.956,Z 403.512,A -85,B 0,C 180,E1 13284.045,E2 13284.045} C_VEL
LIN {X 0,Y 335.325,Z 418.783,A -85,B 0,C 180,E1 13281.832,E2 13281.832} C_VEL
LIN {X 0,Y 336.697,Z 421.898,A -85,B 0,C 180,E1 13281.467,E2 13281.467} C_VEL
LIN {X 0,Y 337.37,Z 437.814,A -85,B 0,C 180,E1 13280.815,E2 13280.815} C_VEL
LIN {X 0,Y 326.808,Z 625.648,A -85,B 0,C 180,E1 13276.582,E2 13276.582} C_VEL
LIN {X 0,Y 324.311,Z 647.5,A -85,B 0,C 180,E1 13275.82,E2 13275.82} C_VEL
LIN {X 0,Y 320.735,Z 668.625,A -85,B 0,C 180,E1 13274.79,E2 13274.79} C_VEL
LIN {X 0,Y 316.617,Z 688.2,A -85,B 0,C 180,E1 13273.504,E2 13273.504} C_VEL
LIN {X 0,Y 312.082,Z 706.941,A -85,B 0,C 180,E1 13271.911,E2 13271.911} C_VEL
LIN {X 0,Y 307.269,Z 724.938,A -85,B 0,C 180,E1 13269.99,E2 13269.99} C_VEL
LIN {X 0,Y 302.301,Z 742.128,A -85,B 0,C 180,E1 13267.725,E2 13267.725} C_VEL
LIN {X 0,Y 297.403,Z 758.44,A -85,B 0,C 180,E1 13265.091,E2 13265.091} C_VEL
LIN {X 0,Y 292.89,Z 773.386,A -85,B 0,C 180,E1 13262.155,E2 13262.155} C_VEL
LIN {X 0,Y 288.865,Z 787.179,A -85,B 0,C 180,E1 13258.871,E2 13258.871} C_VEL
LIN {X 0,Y 285.571,Z 799.569,A -85,B 0,C 180,E1 13255.286,E2 13255.286} C_VEL
LIN {X 0,Y 283.203,Z 810.188,A -85,B 0,C 180,E1 13251.541,E2 13251.541} C_VEL
LIN {X 0,Y 281.699,Z 819.314,A -85,B 0,C 180,E1 13247.559,E2 13247.559} C_VEL
LIN {X 0,Y 281.093,Z 826.462,A -85,B 0,C 180,E1 13243.577,E2 13243.577} C_VEL
LIN {X 0,Y 281.142,Z 831.527,A -85,B 0,C 180,E1 13239.829,E2 13239.829} C_VEL
LIN {X 0,Y 281.522,Z 835.086,A -85,B 0,C 180,E1 13236.042,E2 13236.042} C_VEL
LIN {X 0,Y 281.873,Z 836.875,A -85,B 0,C 180,E1 13232.643,E2 13232.643} C_VEL
LIN {X 0,Y 281.975,Z 837.239,A -85,B 0,C 180,E1 13229.187,E2 13229.187} C_VEL
LIN {X 0,Y 281.742,Z 836.292,A -85,B 0,C 180,E1 13225.93,E2 13225.93} C_VEL
LIN {X 0,Y 281.325,Z 833.649,A -85,B 0,C 180,E1 13222.238,E2 13222.238} C_VEL
LIN {X 0,Y 281.058,Z 829.466,A -85,B 0,C 180,E1 13218.509,E2 13218.509} C_VEL
LIN {X 0,Y 281.291,Z 823.301,A -85,B 0,C 180,E1 13214.539,E2 13214.539} C_VEL
LIN {X 0,Y 282.363,Z 814.738,A -85,B 0,C 180,E1 13210.343,E2 13210.343} C_VEL
LIN {X 0,Y 284.388,Z 804.51,A -85,B 0,C 180,E1 13206.372,E2 13206.372} C_VEL
LIN {X 0,Y 287.337,Z 792.719,A -85,B 0,C 180,E1 13202.657,E2 13202.657} C_VEL
LIN {X 0,Y 290.825,Z 780.243,A -85,B 0,C 180,E1 13199.415,E2 13199.415} C_VEL
LIN {X 0,Y 295.211,Z 765.576,A -85,B 0,C 180,E1 13196.259,E2 13196.259} C_VEL
LIN {X 0,Y 300.035,Z 749.561,A -85,B 0,C 180,E1 13193.429,E2 13193.429} C_VEL
LIN {X 0,Y 305.177,Z 732.071,A -85,B 0,C 180,E1 13190.912,E2 13190.912} C_VEL
LIN {X 0,Y 310.209,Z 713.871,A -85,B 0,C 180,E1 13188.801,E2 13188.801} C_VEL
LIN {X 0,Y 314.895,Z 695.229,A -85,B 0,C 180,E1 13187.073,E2 13187.073} C_VEL
LIN {X 0,Y 319.137,Z 676.11,A -85,B 0,C 180,E1 13185.682,E2 13185.682} C_VEL
LIN {X 0,Y 322.871,Z 656.173,A -85,B 0,C 180,E1 13184.583,E2 13184.583} C_VEL
LIN {X 0,Y 325.768,Z 635.332,A -85,B 0,C 180,E1 13183.739,E2 13183.739} C_VEL
LIN {X 0,Y 327.543,Z 613.548,A -85,B 0,C 180,E1 13183.127,E2 13183.127} C_VEL
LIN {X 0,Y 337.322,Z 435.505,A -85,B 0,C 180,E1 13179.136,E2 13179.136} C_VEL
LIN {X 0,Y 336.383,Z 420.964,A -85,B 0,C 180,E1 13178.487,E2 13178.487} C_VEL
LIN {X 0,Y 327.352,Z 404.292,A -85,B 0,C 180,E1 13176.121,E2 13176.121} C_VEL
LIN {X 0,Y 318.165,Z 389.152,A -85,B 0,C 180,E1 13173.498,E2 13173.498} C_VEL
LIN {X 0,Y 310.074,Z 376.877,A -85,B 0,C 180,E1 13170.952,E2 13170.952} C_VEL
LIN {X 0,Y 307.079,Z 372.3,A -85,B 0,C 180,E1 13169.879,E2 13169.879} C_VEL
LIN {X 0,Y 302.151,Z 362.338,A -85,B 0,C 180,E1 13166.534,E2 13166.534} C_VEL
LIN {X 0,Y 299.009,Z 356.684,A -85,B 0,C 180,E1 13164.286,E2 13164.286} C_VEL
LIN {X 0,Y 297.215,Z 353.057,A -85,B 0,C 180,E1 13162.76,E2 13162.76} C_VEL
LIN {X 0,Y 294.739,Z 348.474,A -85,B 0,C 180,E1 13160.659,E2 13160.659} C_VEL
LIN {X 0,Y 292.419,Z 344.428,A -85,B 0,C 180,E1 13158.541,E2 13158.541} C_VEL
LIN {X 0,Y 291.573,Z 343.125,A -85,B 0,C 180,E1 13157.77,E2 13157.77} C_VEL
LIN {X 0,Y 289.394,Z 339.263,A -85,B 0,C 180,E1 13155.428,E2 13155.428} C_VEL
LIN {X 0,Y 288.505,Z 337.874,A -85,B 0,C 180,E1 13154.449,E2 13154.449} C_VEL
LIN {X 0,Y 286.26,Z 334.378,A -85,B 0,C 180,E1 13151.688,E2 13151.688} C_VEL
LIN {X 0,Y 285.578,Z 332.765,A -85,B 0,C 180,E1 13150.489,E2 13150.489} C_VEL
LIN {X 0,Y 282.527,Z 328.2,A -85,B 0,C 180,E1 13145.075,E2 13145.075} C_VEL
LIN {X 0,Y 282.365,Z 327.333,A -85,B 0,C 180,E1 13143.044,E2 13143.044} C_VEL
LIN {X 0,Y 282.372,Z 327.28,A -85,B 0,C 180,E1 13138.376,E2 13138.376} C_VEL
LIN {X 0,Y 282.353,Z 327.303,A -85,B 0,C 180,E1 13133.697,E2 13133.697} C_VEL
LIN {X 0,Y 282.363,Z 327.302,A -85,B 0,C 180,E1 13128.976,E2 13128.976} C_VEL
LIN {X 0,Y 282.488,Z 327.887,A -85,B 0,C 180,E1 13126.281,E2 13126.281} C_VEL
LIN {X 0,Y 285.785,Z 333.296,A -85,B 0,C 180,E1 13119.948,E2 13119.948} C_VEL
LIN {X 0,Y 287.795,Z 337.273,A -85,B 0,C 180,E1 13116.884,E2 13116.884} C_VEL
LIN {X 0,Y 288.847,Z 338.8,A -85,B 0,C 180,E1 13115.674,E2 13115.674} C_VEL
LIN {X 0,Y 291.137,Z 342.896,A -85,B 0,C 180,E1 13113.042,E2 13113.042} C_VEL
LIN {X 0,Y 294.191,Z 348.88,A -85,B 0,C 180,E1 13109.801,E2 13109.801} C_VEL
LIN {X 0,Y 296.717,Z 353.988,A -85,B 0,C 180,E1 13107.373,E2 13107.373} C_VEL
LIN {X 0,Y 303.78,Z 363.041,A -85,B 0,C 180,E1 13104.599,E2 13104.599} C_VEL
LIN {X 0,Y 311.069,Z 372.839,A -85,B 0,C 180,E1 13102.126,E2 13102.126} C_VEL
LIN {X 0,Y 320.552,Z 386.489,A -85,B 0,C 180,E1 13099.255,E2 13099.255} C_VEL
LIN {X 0,Y 329.948,Z 401.664,A -85,B 0,C 180,E1 13096.685,E2 13096.685} C_VEL
LIN {X 0,Y 336.894,Z 414.244,A -85,B 0,C 180,E1 13094.919,E2 13094.919} C_VEL
LIN {X 0,Y 329.698,Z 570.058,A -85,B 0,C 180,E1 13091.71,E2 13091.71} C_VEL
LIN {X 0,Y 328.353,Z 589.399,A -85,B 0,C 180,E1 13091.039,E2 13091.039} C_VEL
LIN {X 0,Y 326.214,Z 607.713,A -85,B 0,C 180,E1 13090.121,E2 13090.121} C_VEL
LIN {X 0,Y 323.267,Z 625.951,A -85,B 0,C 180,E1 13088.892,E2 13088.892} C_VEL
LIN {X 0,Y 319.625,Z 643.544,A -85,B 0,C 180,E1 13087.363,E2 13087.363} C_VEL
LIN {X 0,Y 315.485,Z 660.029,A -85,B 0,C 180,E1 13085.559,E2 13085.559} C_VEL
LIN {X 0,Y 311.009,Z 675.445,A -85,B 0,C 180,E1 13083.459,E2 13083.459} C_VEL
LIN {X 0,Y 306.307,Z 689.782,A -85,B 0,C 180,E1 13081.047,E2 13081.047} C_VEL
LIN {X 0,Y 301.577,Z 702.968,A -85,B 0,C 180,E1 13078.3,E2 13078.3} C_VEL
LIN {X 0,Y 297.104,Z 714.574,A -85,B 0,C 180,E1 13075.302,E2 13075.302} C_VEL
LIN {X 0,Y 293.064,Z 724.662,A -85,B 0,C 180,E1 13072.042,E2 13072.042} C_VEL
LIN {X 0,Y 289.568,Z 733.237,A -85,B 0,C 180,E1 13068.522,E2 13068.522} C_VEL
LIN {X 0,Y 286.735,Z 740.271,A -85,B 0,C 180,E1 13064.747,E2 13064.747} C_VEL
LIN {X 0,Y 284.752,Z 745.464,A -85,B 0,C 180,E1 13060.93,E2 13060.93} C_VEL
LIN {X 0,Y 283.422,Z 749.138,A -85,B 0,C 180,E1 13056.889,E2 13056.889} C_VEL
LIN {X 0,Y 282.774,Z 751.104,A -85,B 0,C 180,E1 13052.837,E2 13052.837} C_VEL
LIN {X 0,Y 282.67,Z 751.448,A -85,B 0,C 180,E1 13048.784,E2 13048.784} C_VEL
LIN {X 0,Y 283.077,Z 750.186,A -85,B 0,C 180,E1 13044.731,E2 13044.731} C_VEL
LIN {X 0,Y 284.105,Z 747.258,A -85,B 0,C 180,E1 13040.684,E2 13040.684} C_VEL
LIN {X 0,Y 285.762,Z 742.827,A -85,B 0,C 180,E1 13036.855,E2 13036.855} C_VEL
LIN {X 0,Y 288.21,Z 736.649,A -85,B 0,C 180,E1 13033.058,E2 13033.058} C_VEL
LIN {X 0,Y 291.35,Z 728.993,A -85,B 0,C 180,E1 13029.511,E2 13029.511} C_VEL
LIN {X 0,Y 295.262,Z 719.327,A -85,B 0,C 180,E1 13026.024,E2 13026.024} C_VEL
LIN {X 0,Y 299.443,Z 708.736,A -85,B 0,C 180,E1 13022.993,E2 13022.993} C_VEL
LIN {X 0,Y 303.928,Z 696.742,A -85,B 0,C 180,E1 13020.215,E2 13020.215} C_VEL
LIN {X 0,Y 308.75,Z 682.744,A -85,B 0,C 180,E1 13017.592,E2 13017.592} C_VEL
LIN {X 0,Y 313.468,Z 667.529,A -85,B 0,C 180,E1 13015.296,E2 13015.296} C_VEL
LIN {X 0,Y 317.791,Z 651.539,A -85,B 0,C 180,E1 13013.351,E2 13013.351} C_VEL
LIN {X 0,Y 321.723,Z 634.368,A -85,B 0,C 180,E1 13011.684,E2 13011.684} C_VEL
LIN {X 0,Y 324.984,Z 616.61,A -85,B 0,C 180,E1 13010.329,E2 13010.329} C_VEL
LIN {X 0,Y 327.594,Z 597.614,A -85,B 0,C 180,E1 13009.229,E2 13009.229} C_VEL
LIN {X 0,Y 329.331,Z 578.244,A -85,B 0,C 180,E1 13008.429,E2 13008.429} C_VEL
LIN {X 0,Y 330.034,Z 564.642,A -85,B 0,C 180,E1 13008.039,E2 13008.039} C_VEL
LIN {X 0,Y 329.643,Z 557.081,A -85,B 0,C 180,E1 13007.734,E2 13007.734} C_VEL
LIN {X 0,Y 326.126,Z 537.276,A -85,B 0,C 180,E1 13006.549,E2 13006.549} C_VEL
LIN {X 0,Y 325.912,Z 530.757,A -85,B 0,C 180,E1 13006.323,E2 13006.323} C_VEL
LIN {X 0,Y 331.424,Z 417.148,A -85,B 0,C 180,E1 13003.968,E2 13003.968} C_VEL
LIN {X 0,Y 322.089,Z 400.841,A -85,B 0,C 180,E1 13001.452,E2 13001.452} C_VEL
LIN {X 0,Y 313.138,Z 386.861,A -85,B 0,C 180,E1 12998.803,E2 12998.803} C_VEL
LIN {X 0,Y 303.548,Z 373.217,A -85,B 0,C 180,E1 12995.606,E2 12995.606} C_VEL
LIN {X 0,Y 293.892,Z 360.856,A -85,B 0,C 180,E1 12991.883,E2 12991.883} C_VEL
LIN {X 0,Y 289.242,Z 355.015,A -85,B 0,C 180,E1 12989.74,E2 12989.74} C_VEL
LIN {X 0,Y 286.141,Z 348.999,A -85,B 0,C 180,E1 12986.345,E2 12986.345} C_VEL
LIN {X 0,Y 283.721,Z 344.309,A -85,B 0,C 180,E1 12983.248,E2 12983.248} C_VEL
LIN {X 0,Y 281.408,Z 340.402,A -85,B 0,C 180,E1 12979.944,E2 12979.944} C_VEL
LIN {X 0,Y 280.7,Z 339.051,A -85,B 0,C 180,E1 12978.699,E2 12978.699} C_VEL
LIN {X 0,Y 277.789,Z 333.962,A -85,B 0,C 180,E1 12972.05,E2 12972.05} C_VEL
LIN {X 0,Y 276.387,Z 332.628,A -85,B 0,C 180,E1 12966.439,E2 12966.439} C_VEL
LIN {X 0,Y 276.572,Z 332.801,A -85,B 0,C 180,E1 12961.243,E2 12961.243} C_VEL
LIN {X 0,Y 278.076,Z 334.319,A -85,B 0,C 180,E1 12956.29,E2 12956.29} C_VEL
LIN {X 0,Y 281.635,Z 340.034,A -85,B 0,C 180,E1 12949.362,E2 12949.362} C_VEL
LIN {X 0,Y 283.845,Z 344.262,A -85,B 0,C 180,E1 12946.141,E2 12946.141} C_VEL
LIN {X 0,Y 284.804,Z 345.431,A -85,B 0,C 180,E1 12945.151,E2 12945.151} C_VEL
LIN {X 0,Y 287.071,Z 349.665,A -85,B 0,C 180,E1 12942.571,E2 12942.571} C_VEL
LIN {X 0,Y 287.875,Z 350.984,A -85,B 0,C 180,E1 12941.785,E2 12941.785} C_VEL
LIN {X 0,Y 290.746,Z 356.23,A -85,B 0,C 180,E1 12939.044,E2 12939.044} C_VEL
LIN {X 0,Y 293.325,Z 361.286,A -85,B 0,C 180,E1 12936.709,E2 12936.709} C_VEL
LIN {X 0,Y 297.429,Z 368.871,A -85,B 0,C 180,E1 12933.658,E2 12933.658} C_VEL
LIN {X 0,Y 299.486,Z 372.66,A -85,B 0,C 180,E1 12932.405,E2 12932.405} C_VEL
LIN {X 0,Y 308.932,Z 386.315,A -85,B 0,C 180,E1 12929.029,E2 12929.029} C_VEL
LIN {X 0,Y 317.812,Z 400.47,A -85,B 0,C 180,E1 12926.216,E2 12926.216} C_VEL
LIN {X 0,Y 327.251,Z 417.04,A -85,B 0,C 180,E1 12923.513,E2 12923.513} C_VEL
LIN {X 0,Y 331.466,Z 425.611,A -85,B 0,C 180,E1 12922.357,E2 12922.357} C_VEL
LIN {X 0,Y 331.933,Z 439.03,A -85,B 0,C 180,E1 12921.807,E2 12921.807} C_VEL
LIN {X 0,Y 321.091,Z 624.81,A -85,B 0,C 180,E1 12917.585,E2 12917.585} C_VEL
